// TIA Portal V17 program export: 0 tag tables, 0 data types, 22 data blocks, 121 code blocks (in call order from the OBs), 25 instance data blocks

DATA_BLOCK "Reminder"   // DB2
{ S7_Optimized_Access := 'TRUE' }
VERSION : 0.1
// stored: AutoNumber true, DBAccessibleFromOPCUA true, DBAccessibleFromWebserver true, IsOnlyStoredInLoadMemory false, IsRetainMemResEnabled false, IsWriteProtectedInAS false, MemoryReserve 100
   VAR
      x1 : Bool;
   END_VAR
BEGIN
END_DATA_BLOCK

DATA_BLOCK "HMI"   // DB110
{ S7_Optimized_Access := 'TRUE' }
VERSION : 0.1
// stored: AutoNumber false, DBAccessibleFromOPCUA true, DBAccessibleFromWebserver true, IsOnlyStoredInLoadMemory false, IsRetainMemResEnabled false, IsWriteProtectedInAS false, MemoryReserve 100
   VAR
      SS1 : Struct
         xLocalCmd : Bool;
         xEnbCmd : Bool := True;
         xLocalSt : Bool;
         rPacRef : Real;
         rQacRef : Real;
      END_STRUCT;
      SS2 : Struct
         xLocalCmd : Bool;
         xEnbCmd : Bool := True;
         xLocalSt : Bool;
         rPacRef : Real;
         rQacRef : Real;
      END_STRUCT;
      xLocalCmd : Bool;
      xStopCmd : Bool;
      xStandByCmd : Bool;
      xRunCmd : Bool;
      xTestCmd : Bool;
      xLocalSt : Bool;
      xStopSt : Bool;
      xStandBySt : Bool;
      xRunSt : Bool;
      rPacAutomRef : Real;
      PCS1 : Struct
         xEnbDCbus1 : Bool := True;
         xEnbDCbus2 : Bool := True;
      END_STRUCT;
      iNMaxRackFault : Int := 1;
      iNMinRackEnable : Int := 1;
      rSnPE : Real;
      xBB1BR1AlmDisable : Bool;
      xBB1BR2AlmDisable : Bool;
      xBB1BR3AlmDisable : Bool;
      xBB1BR4AlmDisable : Bool;
      xBB1BR5AlmDisable : Bool;
      xBB1BR6AlmDisable : Bool;
      xBB1BR7AlmDisable : Bool;
      xBB1BR8AlmDisable : Bool;
      xBB1BR9AlmDisable : Bool;
      xBB1BR10AlmDisable : Bool;
      xBB2BR1AlmDisable : Bool;
      xBB2BR2AlmDisable : Bool;
      xBB2BR3AlmDisable : Bool;
      xBB2BR4AlmDisable : Bool;
      xBB2BR5AlmDisable : Bool;
      xBB2BR6AlmDisable : Bool;
      xBB2BR7AlmDisable : Bool;
      xBB2BR8AlmDisable : Bool;
      xBB2BR9AlmDisable : Bool;
      xBB2BR10AlmDisable : Bool;
      xBB1AlmDisable : Bool;
      xBB2AlmDisable : Bool;
      xPEMSAlmDisable : Bool;
      xPCSAlmDisable : Bool;
      xMVSkidAlmDisable : Bool;
      xPIAlmDisable : Bool;
   END_VAR
BEGIN
END_DATA_BLOCK

DATA_BLOCK "SM_TEST"   // DB9
{ S7_Optimized_Access := 'TRUE' }
VERSION : 0.1
// stored: AutoNumber true, DBAccessibleFromOPCUA true, DBAccessibleFromWebserver true, IsOnlyStoredInLoadMemory false, IsRetainMemResEnabled false, IsWriteProtectedInAS false, MemoryReserve 100
   VAR
      xEnable_comm : Bool;
      xComm_enabled : Bool;
      xSS1_fault : Bool;
      xAutoCharge_command : Bool;
      xSM1_readyCondition : Bool;
      xSystem_ready : Bool;
      "xBattery_cl/op_command" : Bool;
      xBypass_Estop : Bool;
   END_VAR
BEGIN
END_DATA_BLOCK

DATA_BLOCK "clock"   // DB4
{ S7_Optimized_Access := 'TRUE' }
VERSION : 0.1
// stored: AutoNumber true, DBAccessibleFromOPCUA true, DBAccessibleFromWebserver true, IsOnlyStoredInLoadMemory false, IsRetainMemResEnabled false, IsWriteProtectedInAS false, MemoryReserve 100
   VAR
      xClock_5Hz : Bool;
      xClock_2_5Hz : Bool;
      xClock_2Hz : Bool;
      xClock_1_25Hz : Bool;
      xClock_1Hz : Bool;
      xClock_0_625Hz : Bool;
      xClock_0_5Hz : Bool;
      xClock_10Hz : Bool;
   END_VAR
BEGIN
END_DATA_BLOCK

DATA_BLOCK "BMS1"   // DB21
{ S7_Optimized_Access := 'TRUE' }
VERSION : 0.1
// stored: AutoNumber false, DBAccessibleFromOPCUA true, DBAccessibleFromWebserver true, IsOnlyStoredInLoadMemory false, IsRetainMemResEnabled false, IsWriteProtectedInAS false, MemoryReserve 100
   VAR RETAIN
      TCON { S7_SetPoint := 'True'} : TCON_IP_v4;
   END_VAR
   VAR
      arrData : Array[1..125] of Word;
      xREQ : Bool;
      iCountDone : Int := 1;
      iCountRead : Int := 1;
      MBmode : USInt;
      MBdataAddr : UDInt;
      MBdataLen : UInt;
   END_VAR
   VAR RETAIN
      TCON10 { S7_SetPoint := 'True'} : TCON_IP_v4;
   END_VAR
   VAR
      arrData10 : Array[1..125] of Word;
      xREQ10 : Bool;
      iCountDone10 : Int := 1;
      iCountRead10 : Int := 1;
      MBmode10 : USInt;
      MBdataAddr10 : UDInt;
      MBdataLen10 : UInt;
   END_VAR
   VAR RETAIN
      TCON11 { S7_SetPoint := 'True'} : TCON_IP_v4;
   END_VAR
   VAR
      arrData11 : Array[1..125] of Word;
      xREQ11 : Bool;
      iCountDone11 : Int := 1;
      iCountRead11 : Int := 1;
      MBmode11 : USInt;
      MBdataAddr11 : UDInt;
      MBdataLen11 : UInt;
      BB { S7_SetPoint := 'True'} : "BMS_BB";
      BR01 { S7_SetPoint := 'True'} : "BMS_BR";
      BR02 { S7_SetPoint := 'True'} : "BMS_BR";
      BR03 { S7_SetPoint := 'True'} : "BMS_BR";
      BR04 { S7_SetPoint := 'True'} : "BMS_BR";
      BR05 { S7_SetPoint := 'True'} : "BMS_BR";
      BR06 { S7_SetPoint := 'True'} : "BMS_BR";
      BR07 { S7_SetPoint := 'True'} : "BMS_BR";
      BR08 { S7_SetPoint := 'True'} : "BMS_BR";
      BR09 { S7_SetPoint := 'True'} : "BMS_BR";
      BR10 { S7_SetPoint := 'True'} : "BMS_BR";
      BR11 { S7_SetPoint := 'True'} : "BMS_BR";
      BR12 { S7_SetPoint := 'True'} : "BMS_BR";
      TMS01 { S7_SetPoint := 'True'} : "BMS_TMS";
      TMS02 { S7_SetPoint := 'True'} : "BMS_TMS";
      TMS03 { S7_SetPoint := 'True'} : "BMS_TMS";
      TMS04 { S7_SetPoint := 'True'} : "BMS_TMS";
      TMS05 { S7_SetPoint := 'True'} : "BMS_TMS";
      TMS06 { S7_SetPoint := 'True'} : "BMS_TMS";
      TMS07 { S7_SetPoint := 'True'} : "BMS_TMS";
      TMS08 { S7_SetPoint := 'True'} : "BMS_TMS";
      TMS09 { S7_SetPoint := 'True'} : "BMS_TMS";
      TMS10 { S7_SetPoint := 'True'} : "BMS_TMS";
      TMS11 { S7_SetPoint := 'True'} : "BMS_TMS";
      TMS12 { S7_SetPoint := 'True'} : "BMS_TMS";
      rNomEnergyBank { S7_SetPoint := 'True'} : Real;
      rPbank : Real;
      rCrate : Real;
      rSOCavlCha : Real;
      rSOCavlDsch : Real;
      rEnergyAvlCha : Real;
      rEnergyAvlDsch : Real;
      diTimeEndCha : DInt;
      diTimeEndDsch : DInt;
      rVcellMinSet : Real := 2.76;
      rVcellMinReset : Real := 3.05;
      rVcellMaxSet : Real := 3.68;
      rVcellMaxReset : Real := 3.3;
      rVcellAutoChaSet : Real := 2.7;
      rVcellAutoChaReset : Real := 3.1;
      rPchaLim : Real;
      rPdschLim : Real;
      wRackFlt : Word;
      wRackOn : Word;
      xBankAvl : Bool;
      xEnbCha : Bool;
      xEnbDsch : Bool;
      xAutoChaCmd : Bool;
      xSwitchGearSt : Bool;
      xPwrOffReadySt : Bool;
      xPwrOnReadySt : Bool;
      xPwrOnFltSt : Bool;
      xPwrOffFltSt : Bool;
      xInitSt : Bool;
      xNormOpSt : Bool;
      xFullChaSt : Bool;
      xFullDschSt : Bool;
      xWarnSt : Bool;
      xFltSt : Bool;
      xInitCmd : Bool;
      xStayCmd : Bool;
      xCloseCmd : Bool;
      xOpenCmd : Bool;
      xFltClearCmd : Bool;
      wCmd : Word;
      wFltClearCmd : Word;
      BBwAlm1 : Word;
      BBwWarn1 : Word;
      BBxCommFltSt : Bool;
      BBxFltSt : Bool;
      BBxAlmSt : Bool;
      BBxWarnSt : Bool;
      BR01wAlm1 : Word;
      BR01wAlm2 : Word;
      BR01wAlm3 : Word;
      BR01wWarn1 : Word;
      BR01xFltSt : Bool;
      BR01xAlmSt : Bool;
      BR01xWarnSt : Bool;
      BR02wAlm1 : Word;
      BR02wAlm2 : Word;
      BR02wAlm3 : Word;
      BR02wWarn1 : Word;
      BR02xFltSt : Bool;
      BR02xAlmSt : Bool;
      BR02xWarnSt : Bool;
      BR03wAlm1 : Word;
      BR03wAlm2 : Word;
      BR03wAlm3 : Word;
      BR03wWarn1 : Word;
      BR03xFltSt : Bool;
      BR03xAlmSt : Bool;
      BR03xWarnSt : Bool;
      BR04wAlm1 : Word;
      BR04wAlm2 : Word;
      BR04wAlm3 : Word;
      BR04wWarn1 : Word;
      BR04xFltSt : Bool;
      BR04xAlmSt : Bool;
      BR04xWarnSt : Bool;
      BR05wAlm1 : Word;
      BR05wAlm2 : Word;
      BR05wAlm3 : Word;
      BR05wWarn1 : Word;
      BR05xFltSt : Bool;
      BR05xAlmSt : Bool;
      BR05xWarnSt : Bool;
      BR06wAlm1 : Word;
      BR06wAlm2 : Word;
      BR06wAlm3 : Word;
      BR06wWarn1 : Word;
      BR06xFltSt : Bool;
      BR06xAlmSt : Bool;
      BR06xWarnSt : Bool;
      BR07wAlm1 : Word;
      BR07wAlm2 : Word;
      BR07wAlm3 : Word;
      BR07wWarn1 : Word;
      BR07xFltSt : Bool;
      BR07xAlmSt : Bool;
      BR07xWarnSt : Bool;
      BR08wAlm1 : Word;
      BR08wAlm2 : Word;
      BR08wAlm3 : Word;
      BR08wWarn1 : Word;
      BR08xFltSt : Bool;
      BR08xAlmSt : Bool;
      BR08xWarnSt : Bool;
      BR09wAlm1 : Word;
      BR09wAlm2 : Word;
      BR09wAlm3 : Word;
      BR09wWarn1 : Word;
      BR09xFltSt : Bool;
      BR09xAlmSt : Bool;
      BR09xWarnSt : Bool;
      BR10wAlm1 : Word;
      BR10wAlm2 : Word;
      BR10wAlm3 : Word;
      BR10wWarn1 : Word;
      BR10xFltSt : Bool;
      BR10xAlmSt : Bool;
      BR10xWarnSt : Bool;
      BR11wAlm1 : Word;
      BR11wAlm2 : Word;
      BR11wAlm3 : Word;
      BR11wWarn1 : Word;
      BR11xFltSt : Bool;
      BR11xAlmSt : Bool;
      BR11xWarnSt : Bool;
      BR12wAlm1 : Word;
      BR12wAlm2 : Word;
      BR12wAlm3 : Word;
      BR12wWarn1 : Word;
      BR12xFltSt : Bool;
      BR12xAlmSt : Bool;
      BR12xWarnSt : Bool;
      iNRackFault : Int;
      BR01xSSFltSt : Bool;
      BR02xSSFltSt : Bool;
      BR03xSSFltSt : Bool;
      BR04xSSFltSt : Bool;
      BR05xSSFltSt : Bool;
      BR06xSSFltSt : Bool;
      BR07xSSFltSt : Bool;
      BR08xSSFltSt : Bool;
      BR09xSSFltSt : Bool;
      BR10xSSFltSt : Bool;
      BR11xSSFltSt : Bool;
      BR12xSSFltSt : Bool;
   END_VAR
BEGIN
   TCON.RemoteAddress.ADDR[1] := 192;
   TCON.RemoteAddress.ADDR[2] := 168;
   TCON.RemoteAddress.ADDR[3] := 150;
   TCON.RemoteAddress.ADDR[4] := 44;
   TCON10.RemoteAddress.ADDR[1] := 192;
   TCON10.RemoteAddress.ADDR[2] := 168;
   TCON10.RemoteAddress.ADDR[3] := 150;
   TCON10.RemoteAddress.ADDR[4] := 44;
   TCON11.RemoteAddress.ADDR[1] := 192;
   TCON11.RemoteAddress.ADDR[2] := 168;
   TCON11.RemoteAddress.ADDR[3] := 150;
   TCON11.RemoteAddress.ADDR[4] := 44;
   BB.iNBRtotalCount := 10;
END_DATA_BLOCK

DATA_BLOCK "BMS2"   // DB22
{ S7_Optimized_Access := 'TRUE' }
VERSION : 0.1
// stored: AutoNumber false, DBAccessibleFromOPCUA true, DBAccessibleFromWebserver true, IsOnlyStoredInLoadMemory false, IsRetainMemResEnabled false, IsWriteProtectedInAS false, MemoryReserve 100
   VAR RETAIN
      TCON { S7_SetPoint := 'True'} : TCON_IP_v4;
   END_VAR
   VAR
      arrData : Array[1..125] of Word;
      xREQ : Bool;
      iCountDone : Int := 1;
      iCountRead : Int := 1;
      MBmode : USInt;
      MBdataAddr : UDInt;
      MBdataLen : UInt;
   END_VAR
   VAR RETAIN
      TCON10 { S7_SetPoint := 'True'} : TCON_IP_v4;
   END_VAR
   VAR
      arrData10 : Array[1..125] of Word;
      xREQ10 : Bool;
      iCountDone10 : Int := 1;
      iCountRead10 : Int := 1;
      MBmode10 : USInt;
      MBdataAddr10 : UDInt;
      MBdataLen10 : UInt;
   END_VAR
   VAR RETAIN
      TCON11 { S7_SetPoint := 'True'} : TCON_IP_v4;
   END_VAR
   VAR
      arrData11 : Array[1..125] of Word;
      xREQ11 : Bool;
      iCountDone11 : Int := 1;
      iCountRead11 : Int := 1;
      MBmode11 : USInt;
      MBdataAddr11 : UDInt;
      MBdataLen11 : UInt;
      BB { S7_SetPoint := 'True'} : "BMS_BB";
      BR01 { S7_SetPoint := 'True'} : "BMS_BR";
      BR02 { S7_SetPoint := 'True'} : "BMS_BR";
      BR03 { S7_SetPoint := 'True'} : "BMS_BR";
      BR04 { S7_SetPoint := 'True'} : "BMS_BR";
      BR05 { S7_SetPoint := 'True'} : "BMS_BR";
      BR06 { S7_SetPoint := 'True'} : "BMS_BR";
      BR07 { S7_SetPoint := 'True'} : "BMS_BR";
      BR08 { S7_SetPoint := 'True'} : "BMS_BR";
      BR09 { S7_SetPoint := 'True'} : "BMS_BR";
      BR10 { S7_SetPoint := 'True'} : "BMS_BR";
      TMS01 { S7_SetPoint := 'True'} : "BMS_TMS";
      TMS02 { S7_SetPoint := 'True'} : "BMS_TMS";
      TMS03 { S7_SetPoint := 'True'} : "BMS_TMS";
      TMS04 { S7_SetPoint := 'True'} : "BMS_TMS";
      TMS05 { S7_SetPoint := 'True'} : "BMS_TMS";
      TMS06 { S7_SetPoint := 'True'} : "BMS_TMS";
      TMS07 { S7_SetPoint := 'True'} : "BMS_TMS";
      TMS08 { S7_SetPoint := 'True'} : "BMS_TMS";
      TMS09 { S7_SetPoint := 'True'} : "BMS_TMS";
      TMS10 { S7_SetPoint := 'True'} : "BMS_TMS";
      rNomEnergyBank { S7_SetPoint := 'True'} : Real;
      rPbank : Real;
      rCrate : Real;
      rSOCavlCha : Real;
      rSOCavlDsch : Real;
      rEnergyAvlCha : Real;
      rEnergyAvlDsch : Real;
      diTimeEndCha : DInt;
      diTimeEndDsch : DInt;
      rVcellMinSet : Real := 2.76;
      rVcellMinReset : Real := 3.05;
      rVcellMaxSet : Real := 3.68;
      rVcellMaxReset : Real := 3.3;
      rVcellAutoChaSet : Real := 2.7;
      rVcellAutoChaReset : Real := 3.1;
      rPchaLim : Real;
      rPdschLim : Real;
      wRackFlt : Word;
      wRackOn : Word;
      xBankAvl : Bool;
      xEnbCha : Bool;
      xEnbDsch : Bool;
      xAutoChaCmd : Bool;
      xSwitchGearSt : Bool;
      xPwrOffReadySt : Bool;
      xPwrOnReadySt : Bool;
      xPwrOnFltSt : Bool;
      xPwrOffFltSt : Bool;
      xInitSt : Bool;
      xNormOpSt : Bool;
      xFullChaSt : Bool;
      xFullDschSt : Bool;
      xWarnSt : Bool;
      xFltSt : Bool;
      xInitCmd : Bool;
      xStayCmd : Bool;
      xCloseCmd : Bool;
      xOpenCmd : Bool;
      xFltClearCmd : Bool;
      wCmd : Word;
      wFltClearCmd : Word;
      BBwAlm1 : Word;
      BBwWarn1 : Word;
      BBxCommFltSt : Bool;
      BBxFltSt : Bool;
      BBxAlmSt : Bool;
      BBxWarnSt : Bool;
      BR01wAlm1 : Word;
      BR01wAlm2 : Word;
      BR01wAlm3 : Word;
      BR01wWarn1 : Word;
      BR01xFltSt : Bool;
      BR01xAlmSt : Bool;
      BR01xWarnSt : Bool;
      BR02wAlm1 : Word;
      BR02wAlm2 : Word;
      BR02wAlm3 : Word;
      BR02wWarn1 : Word;
      BR02xFltSt : Bool;
      BR02xAlmSt : Bool;
      BR02xWarnSt : Bool;
      BR03wAlm1 : Word;
      BR03wAlm2 : Word;
      BR03wAlm3 : Word;
      BR03wWarn1 : Word;
      BR03xFltSt : Bool;
      BR03xAlmSt : Bool;
      BR03xWarnSt : Bool;
      BR04wAlm1 : Word;
      BR04wAlm2 : Word;
      BR04wAlm3 : Word;
      BR04wWarn1 : Word;
      BR04xFltSt : Bool;
      BR04xAlmSt : Bool;
      BR04xWarnSt : Bool;
      BR05wAlm1 : Word;
      BR05wAlm2 : Word;
      BR05wAlm3 : Word;
      BR05wWarn1 : Word;
      BR05xFltSt : Bool;
      BR05xAlmSt : Bool;
      BR05xWarnSt : Bool;
      BR06wAlm1 : Word;
      BR06wAlm2 : Word;
      BR06wAlm3 : Word;
      BR06wWarn1 : Word;
      BR06xFltSt : Bool;
      BR06xAlmSt : Bool;
      BR06xWarnSt : Bool;
      BR07wAlm1 : Word;
      BR07wAlm2 : Word;
      BR07wAlm3 : Word;
      BR07wWarn1 : Word;
      BR07xFltSt : Bool;
      BR07xAlmSt : Bool;
      BR07xWarnSt : Bool;
      BR08wAlm1 : Word;
      BR08wAlm2 : Word;
      BR08wAlm3 : Word;
      BR08wWarn1 : Word;
      BR08xFltSt : Bool;
      BR08xAlmSt : Bool;
      BR08xWarnSt : Bool;
      BR09wAlm1 : Word;
      BR09wAlm2 : Word;
      BR09wAlm3 : Word;
      BR09wWarn1 : Word;
      BR09xFltSt : Bool;
      BR09xAlmSt : Bool;
      BR09xWarnSt : Bool;
      BR10wAlm1 : Word;
      BR10wAlm2 : Word;
      BR10wAlm3 : Word;
      BR10wWarn1 : Word;
      BR10xFltSt : Bool;
      BR10xAlmSt : Bool;
      BR10xWarnSt : Bool;
      iNRackFault : Int;
      BR01xSSFltSt : Bool;
      BR02xSSFltSt : Bool;
      BR03xSSFltSt : Bool;
      BR04xSSFltSt : Bool;
      BR05xSSFltSt : Bool;
      BR06xSSFltSt : Bool;
      BR07xSSFltSt : Bool;
      BR08xSSFltSt : Bool;
      BR09xSSFltSt : Bool;
      BR10xSSFltSt : Bool;
   END_VAR
BEGIN
   TCON.RemoteAddress.ADDR[1] := 192;
   TCON.RemoteAddress.ADDR[2] := 168;
   TCON.RemoteAddress.ADDR[3] := 150;
   TCON.RemoteAddress.ADDR[4] := 44;
   TCON10.RemoteAddress.ADDR[1] := 192;
   TCON10.RemoteAddress.ADDR[2] := 168;
   TCON10.RemoteAddress.ADDR[3] := 150;
   TCON10.RemoteAddress.ADDR[4] := 44;
   TCON11.RemoteAddress.ADDR[1] := 192;
   TCON11.RemoteAddress.ADDR[2] := 168;
   TCON11.RemoteAddress.ADDR[3] := 150;
   TCON11.RemoteAddress.ADDR[4] := 44;
   BB.iNBRtotalCount := 10;
END_DATA_BLOCK

DATA_BLOCK "EME"   // DB502, F_DB
{ S7_Optimized_Access := 'TRUE' }
VERSION : 0.1
// stored: AutoNumber false, DBAccessibleFromOPCUA true, DBAccessibleFromWebserver true
   VAR
      xAlwaysOff : Bool;
      xBattOpenCmd : Bool;
      xStopPCSCmd : Bool;
      xMVbrkOpenCmd : Bool;
      xMVtrafoSt : Bool;
      xAuxSkid : Bool;
      xAuxSkidDelay : Bool;
      xAuxSkidFireMan : Bool;
      xAuxSkidFireManDelay : Bool;
      xCore : Bool;
      xCoreDelay : Bool;
      xTwinPCS : Bool;
      xPCSCmd : Bool;
      xResetCmd : Bool;
      xByPass : Bool;
      xRcvError : Bool;
      xSendError : Bool;
      xAckReq : Bool;
      xByPassCore : Bool;
   END_VAR
BEGIN
END_DATA_BLOCK

DATA_BLOCK "Emergency_DB"   // DB502, F_DB
{ S7_Optimized_Access := 'TRUE' }
VERSION : 0.1
// stored: AutoNumber false, DBAccessibleFromOPCUA true, DBAccessibleFromWebserver true
   VAR
      xAlwaysOff : Bool;
      xBattOpenCmd : Bool;
      xStopPCSCmd : Bool;
      xMVbrkOpenCmd : Bool;
      xMVtrafoSt : Bool;
      xAuxSkid : Bool;
      xAuxSkidDelay : Bool;
      xAuxSkidFireMan : Bool;
      xAuxSkidFireManDelay : Bool;
      xCore : Bool;
      xCoreDelay : Bool;
      xTwinPCS : Bool;
      xPCSCmd : Bool;
      xResetCmd : Bool;
      xByPass : Bool;
      xRcvError : Bool;
      xSendError : Bool;
      xAckReq : Bool;
      xByPassCore : Bool;
      xTripPemsBattery : Bool;
   END_VAR
BEGIN
END_DATA_BLOCK

DATA_BLOCK "SM1"   // DB61
{ S7_Optimized_Access := 'TRUE' }
VERSION : 0.1
// stored: AutoNumber false, DBAccessibleFromOPCUA true, DBAccessibleFromWebserver true, IsOnlyStoredInLoadMemory false, IsRetainMemResEnabled false, IsWriteProtectedInAS false, MemoryReserve 100
   VAR
      xT11 : Bool;
      xT21 : Bool;
      xT22 : Bool;
      xT31 : Bool;
      xT32 : Bool;
      xT33 : Bool;
      xT34 : Bool;
      xT41 : Bool;
      xT42 : Bool;
      xT43 : Bool;
      xT44 : Bool;
      xT51 : Bool;
      xT52 : Bool;
      xT53 : Bool;
      xT61 : Bool;
      xT62 : Bool;
      xT71 : Bool;
      xT72 : Bool;
      xT73 : Bool;
      xT81 : Bool;
      xT91 : Bool;
      xSsBootSt : Bool;
      xSsWarmUpSt : Bool;
      xSsReadySt : Bool;
      xSsStandBySt : Bool;
      xSsRunSt : Bool;
      xSsTestSt : Bool;
      xSsAutoMaintSt : Bool;
      xSsStopSt : Bool;
      xSsFaultSt : Bool;
      iCountSS : Int;
      xBootSt : Bool;
      xRunPlcSt : Bool;
      xCommCmd : Bool;
      xAuxCmd : Bool;
      xCommSt : Bool;
      xAuxSt : Bool;
      xFltSt : Bool;
      xEnbSSysSt : Bool;
      xReadyCondSt : Bool;
      xTestCmd : Bool;
      xBattCloseCmd : Bool;
      xBattCloseSt : Bool;
      xBattOpenSt : Bool;
      xStopCmd : Bool;
      xStandByCmd : Bool;
      xAutomaintCmd : Bool;
      xStopAutomaintCmd : Bool;
      xAutomaintSt : Bool;
      xRunCmd : Bool;
      xPCSenbCmd : Bool;
      xPCSrunCmd : Bool;
      xMVbreakerCloseSt : Bool;
      xPCSrunSt : Bool;
      xPCSstopSt : Bool;
      xPCSreadySt : Bool;
      rPacAutomRef : Real;
      xVacPCS : Bool;
      xMVbreakerOpenCmd : Bool;
      xMVbreakerOpenSt : Bool;
   END_VAR
BEGIN
END_DATA_BLOCK

DATA_BLOCK "SM2"   // DB71
{ S7_Optimized_Access := 'TRUE' }
VERSION : 0.1
// stored: AutoNumber false, DBAccessibleFromOPCUA true, DBAccessibleFromWebserver true, IsOnlyStoredInLoadMemory false, IsRetainMemResEnabled false, IsWriteProtectedInAS false, MemoryReserve 100
   VAR
      xT11 : Bool;
      xT21 : Bool;
      xT22 : Bool;
      xT31 : Bool;
      xT32 : Bool;
      xT33 : Bool;
      xT34 : Bool;
      xT41 : Bool;
      xT42 : Bool;
      xT43 : Bool;
      xT44 : Bool;
      xT51 : Bool;
      xT52 : Bool;
      xT53 : Bool;
      xT61 : Bool;
      xT62 : Bool;
      xT71 : Bool;
      xT72 : Bool;
      xT73 : Bool;
      xT81 : Bool;
      xT91 : Bool;
      xSsBootSt : Bool;
      xSsWarmUpSt : Bool;
      xSsReadySt : Bool;
      xSsStandBySt : Bool;
      xSsRunSt : Bool;
      xSsTestSt : Bool;
      xSsAutoMaintSt : Bool;
      xSsStopSt : Bool;
      xSsFaultSt : Bool;
      iCountSS : Int;
      xBootSt : Bool;
      xRunPlcSt : Bool;
      xCommCmd : Bool;
      xAuxCmd : Bool;
      xCommSt : Bool;
      xAuxSt : Bool;
      xFltSt : Bool;
      xEnbSSysSt : Bool;
      xReadyCondSt : Bool;
      xTestCmd : Bool;
      xBattCloseCmd : Bool;
      xBattCloseSt : Bool;
      xBattOpenSt : Bool;
      xStopCmd : Bool;
      xStandByCmd : Bool;
      xAutomaintCmd : Bool;
      xStopAutomaintCmd : Bool;
      xAutomaintSt : Bool;
      xRunCmd : Bool;
      xPCSenbCmd : Bool;
      xPCSrunCmd : Bool;
      xMVbreakerCloseSt : Bool;
      xPCSrunSt : Bool;
      xPCSstopSt : Bool;
      xPCSreadySt : Bool;
      rPacAutomRef : Real;
      xVacPCS : Bool;
      xMVbreakerOpenCmd : Bool;
      xMVbreakerOpenSt : Bool;
   END_VAR
BEGIN
END_DATA_BLOCK

DATA_BLOCK "SS"   // DB101
{ S7_Optimized_Access := 'TRUE' }
VERSION : 0.1
// stored: AutoNumber false, DBAccessibleFromOPCUA true, DBAccessibleFromWebserver true, IsOnlyStoredInLoadMemory false, IsRetainMemResEnabled false, IsWriteProtectedInAS false, MemoryReserve 100
   VAR
      xFltSt : Bool;
      xSs1FltSt : Bool;
      xSs2FltSt : Bool;
      xAlmSt : Bool;
      XWarSt : Bool;   // Warning status
      wAlm1 : Word;
      wAlm2 : Word;
      wAlm3 : Word;
      wAlm4 : Word;
      wAlm5 : Word;
      wWarn1 : Word;
      wWarn2 : Word;
      wWarn3 : Word;
      wWarn4 : Word;
      wWarn5 : Word;
   END_VAR
BEGIN
END_DATA_BLOCK

DATA_BLOCK "DigitalOutput_DB"   // DB1
{ S7_Optimized_Access := 'TRUE' }
VERSION : 0.1
// stored: AutoNumber true, DBAccessibleFromOPCUA true, DBAccessibleFromWebserver true, IsOnlyStoredInLoadMemory false, IsRetainMemResEnabled false, IsWriteProtectedInAS false, MemoryReserve 100
   VAR
      xEnable : Bool;
   END_VAR
BEGIN
END_DATA_BLOCK

DATA_BLOCK "DashBoard"   // DB121
{ S7_Optimized_Access := 'FALSE' }
VERSION : 0.1
// stored: AutoNumber false, DBAccessibleFromOPCUA true, DBAccessibleFromWebserver true, IsOnlyStoredInLoadMemory false, IsWriteProtectedInAS false
   VAR
      BB1 { S7_SetPoint := 'True'} : "BB";
      BB2 { S7_SetPoint := 'True'} : "BB";
      BB1BR1 : "BR";
      BB1BR2 : "BR";
      BB1BR3 : "BR";
      BB1BR4 : "BR";
      BB1BR5 : "BR";
      BB1BR6 : "BR";
      BB1BR7 : "BR";
      BB1BR8 : "BR";
      BB1BR9 : "BR";
      BB1BR10 : "BR";
      BB1BR11 : "BR";
      BB1BR12 : "BR";
      BB2BR1 : "BR";
      BB2BR2 : "BR";
      BB2BR3 : "BR";
      BB2BR4 : "BR";
      BB2BR5 : "BR";
      BB2BR6 : "BR";
      BB2BR7 : "BR";
      BB2BR8 : "BR";
      BB2BR9 : "BR";
      BB2BR10 : "BR";
      BB2BR11 : "BR";
      BB2BR12 : "BR";
      PCS : "PCS";
      MVSKID { S7_SetPoint := 'True'} : "MVSKID";
      SM { S7_SetPoint := 'True'} : "SM";
   END_VAR
BEGIN
END_DATA_BLOCK

DATA_BLOCK "ED"   // DB400
{ S7_Optimized_Access := 'TRUE' }
VERSION : 0.1
// stored: AutoNumber false, DBAccessibleFromOPCUA true, DBAccessibleFromWebserver true, IsOnlyStoredInLoadMemory false, IsRetainMemResEnabled false, IsWriteProtectedInAS false, MemoryReserve 100
   VAR
      Pems : Struct
         LinkState : Array[1..52] of "LPNDR_typePortLinkState";
         X1 : Bool;
         X2 : Bool;
         X3 : Bool;
      END_STRUCT;
      ET200 : Struct
         LinkState : Array[1..52] of "LPNDR_typePortLinkState";
         X1 : Bool;
         X2 : Bool;
      END_STRUCT;
   END_VAR
BEGIN
END_DATA_BLOCK

DATA_BLOCK "NTPserver"   // DB122
{ S7_Optimized_Access := 'TRUE' }
VERSION : 0.1
// stored: AutoNumber false, DBAccessibleFromOPCUA true, DBAccessibleFromWebserver true, IsOnlyStoredInLoadMemory false, IsRetainMemResEnabled false, IsWriteProtectedInAS false, MemoryReserve 100
   VAR
      x_lEnable : Bool := true;
      i_Reference : USInt;
      dtl_Time : DTL;
      i_auxRetVal : Int;
   END_VAR
BEGIN
END_DATA_BLOCK

DATA_BLOCK "MV SKID"   // DB42
{ S7_Optimized_Access := 'TRUE' }
VERSION : 0.1
// stored: AutoNumber false, DBAccessibleFromOPCUA true, DBAccessibleFromWebserver true, IsOnlyStoredInLoadMemory false, IsRetainMemResEnabled false, IsWriteProtectedInAS false, MemoryReserve 100
   VAR RETAIN
      TCON { S7_SetPoint := 'True'} : TCON_IP_v4;
   END_VAR
   VAR
      arrData : Array[1..125] of Word;
      xREQ : Bool;
      iCountDone : Int := 1;
      iCountRead : Int := 1;
      MBmode : USInt;
      MBdataAddr : UDInt;
      MBdataLen : UInt;
      R : "R_MV";
      W { S7_SetPoint := 'True'} : "W_MV";
      xFltSt { S7_SetPoint := 'True'} : Bool;
      xAlmSt : Bool;
      xWarnSt : Bool;
      wLine1DiscSt : Word;
      wLine2DiscSt : Word;
      wProt1DiscSt : Word;
      wProt1CircBrkSt : Word;
   END_VAR
BEGIN
   TCON.RemoteAddress.ADDR[1] := 192;
   TCON.RemoteAddress.ADDR[2] := 168;
   TCON.RemoteAddress.ADDR[3] := 150;
   TCON.RemoteAddress.ADDR[4] := 44;
END_DATA_BLOCK

DATA_BLOCK "MvSkid_1"   // DB42
{ S7_Optimized_Access := 'TRUE' }
VERSION : 0.1
// stored: AutoNumber false, DBAccessibleFromOPCUA true, DBAccessibleFromWebserver true, IsOnlyStoredInLoadMemory false, IsRetainMemResEnabled false, IsWriteProtectedInAS false, MemoryReserve 100
   VAR RETAIN
      TCON { S7_SetPoint := 'True'} : TCON_IP_v4;
   END_VAR
   VAR
      arrData : Array[1..125] of Word;
      xREQ : Bool;
      iCountRead : Int := 1;
      MBmode : USInt;
      MBdataAddr : UDInt;
      MBdataLen : UInt;
      R : "R_MV";
      iCountDone : Int := 1;
      W { S7_SetPoint := 'True'} : "W_MV";
      xFltSt { S7_SetPoint := 'True'} : Bool;
      xAlmSt : Bool;
      xWarnSt : Bool;
      wLine1DiscSt : Word;
      wLine2DiscSt : Word;
      wProt1DiscSt : Word;
      wProt1CircBrkSt : Word;
   END_VAR
BEGIN
   TCON.RemoteAddress.ADDR[1] := 192;
   TCON.RemoteAddress.ADDR[2] := 168;
   TCON.RemoteAddress.ADDR[3] := 150;
   TCON.RemoteAddress.ADDR[4] := 44;
END_DATA_BLOCK

DATA_BLOCK "MvSkid_2"   // DB46
{ S7_Optimized_Access := 'TRUE' }
VERSION : 0.1
// stored: AutoNumber true, DBAccessibleFromOPCUA true, DBAccessibleFromWebserver true, IsOnlyStoredInLoadMemory false, IsRetainMemResEnabled false, IsWriteProtectedInAS false, MemoryReserve 100
   VAR RETAIN
      TCON { S7_SetPoint := 'True'} : TCON_IP_v4;
   END_VAR
   VAR
      arrData : Array[1..125] of Word;
      xREQ : Bool;
      iCountDone : Int := 1;
      iCountRead : Int := 1;
      MBmode : USInt;
      MBdataAddr : UDInt;
      MBdataLen : UInt;
      R : "R_MV";
      W { S7_SetPoint := 'True'} : "W_MV";
      xFltSt { S7_SetPoint := 'True'} : Bool;
      xAlmSt : Bool;
      xWarnSt : Bool;
      wLine1DiscSt : Word;
      wLine2DiscSt : Word;
      wProt1DiscSt : Word;
      wProt1CircBrkSt : Word;
   END_VAR
BEGIN
   TCON.RemoteAddress.ADDR[1] := 192;
   TCON.RemoteAddress.ADDR[2] := 168;
   TCON.RemoteAddress.ADDR[3] := 150;
   TCON.RemoteAddress.ADDR[4] := 44;
END_DATA_BLOCK

DATA_BLOCK "PCS1"   // DB41
{ S7_Optimized_Access := 'TRUE' }
VERSION : 0.1
// stored: AutoNumber false, DBAccessibleFromOPCUA true, DBAccessibleFromWebserver true, IsOnlyStoredInLoadMemory false, IsRetainMemResEnabled false, IsWriteProtectedInAS false, MemoryReserve 100
   VAR RETAIN
      TCON { S7_SetPoint := 'True'} : TCON_IP_v4;
   END_VAR
   VAR
      arrData : Array[1..125] of Word;
      xREQ : Bool;
      iCountDone : Int := 1;
      iCountRead : Int := 1;
      MBmode : USInt;
      MBdataAddr : UDInt;
      MBdataLen : UInt;
   END_VAR
   VAR RETAIN
      TCON10 { S7_SetPoint := 'True'} : TCON_IP_v4;
   END_VAR
   VAR
      arrData10 : Array[1..125] of Word;
      xREQ10 : Bool;
      iCountDone10 : Int := 1;
      iCountRead10 : Int := 1;
      MBmode10 : USInt;
      MBdataAddr10 : UDInt;
      MBdataLen10 : UInt;
      R { S7_SetPoint := 'True'} : "R_PE";
      RW { S7_SetPoint := 'True'} : "RW_PE";
      W { S7_SetPoint := 'True'} : "W_PE";
   END_VAR
   VAR RETAIN
      TCONW { S7_SetPoint := 'True'} : TCON_IP_v4;
   END_VAR
   VAR
      arrDataW : Array[1..125] of Word;
      xREQW : Bool;
      iCountDoneW : Int := 1;
      iCountReadW : Int := 1;
      MBmodeW : USInt;
      MBdataAddrW : UDInt;
      MBdataLenW : UInt;
      xDCbus1Avl : Bool;
      xDCbus2Avl : Bool;
      xLVRT : Bool;
      xOVRT : Bool;
      xCommFltSt : Bool;
      xFltSt : Bool;
      xWarnSt : Bool;
      xModFltBus1St : Bool;
      xModFltBus2St : Bool;
      xMod1FltSt : Bool;
      xMod2FltSt : Bool;
      xMod3FltSt : Bool;
      xMod4FltSt : Bool;
      xMod5FltSt : Bool;
      xMod6FltSt : Bool;
      xMod1WarnSt : Bool;
      xMod2WarnSt : Bool;
      xMod3WarnSt : Bool;
      xMod4WarnSt : Bool;
      xMod5WarnSt : Bool;
      xMod6WarnSt : Bool;
      rMod1MaxTemp : Real;
      rMod2MaxTemp : Real;
      rMod3MaxTemp : Real;
      rMod4MaxTemp : Real;
      rMod5MaxTemp : Real;
      rMod6MaxTemp : Real;
      rPacBus1Meas : Real;
      rPacBus2Meas : Real;
      rQacBus1Meas : Real;
      rQacBus2Meas : Real;
      rVacMeas : Real;
      rIacTotMeas : Real;
      iCodeFlt : Int;
      iCodeWarn : Int;
      iModFlt : Int;
      iModWarn : Int;
      wInvFlt1 : Word;
      wInvFlt2 : Word;
      wInvFlt3 : Word;
      wInvFlt4 : Word;
      wInvFlt5 : Word;
      wInvFlt6 : Word;
      wInvFlt7 : Word;
      wInvWarn1 : Word;
      wInvWarn2 : Word;
      wInvWarn3 : Word;
      wInvWarn4 : Word;
      wInvWarn5 : Word;
      wInvWarn6 : Word;
      wMod1Flt1 : Word;
      wMod1Flt2 : Word;
      wMod1Flt3 : Word;
      wMod1Flt4 : Word;
      wMod2Flt1 : Word;
      wMod2Flt2 : Word;
      wMod2Flt3 : Word;
      wMod2Flt4 : Word;
      wMod3Flt1 : Word;
      wMod3Flt2 : Word;
      wMod3Flt3 : Word;
      wMod3Flt4 : Word;
      wMod4Flt1 : Word;
      wMod4Flt2 : Word;
      wMod4Flt3 : Word;
      wMod4Flt4 : Word;
      wMod5Flt1 : Word;
      wMod5Flt2 : Word;
      wMod5Flt3 : Word;
      wMod5Flt4 : Word;
      wMod6Flt1 : Word;
      wMod6Flt2 : Word;
      wMod6Flt3 : Word;
      wMod6Flt4 : Word;
      wMod1Warn1 : Word;
      wMod1Warn2 : Word;
      wMod1Warn3 : Word;
      wMod1Warn4 : Word;
      wMod2Warn1 : Word;
      wMod2Warn2 : Word;
      wMod2Warn3 : Word;
      wMod2Warn4 : Word;
      wMod3Warn1 : Word;
      wMod3Warn2 : Word;
      wMod3Warn3 : Word;
      wMod3Warn4 : Word;
      wMod4Warn1 : Word;
      wMod4Warn2 : Word;
      wMod4Warn3 : Word;
      wMod4Warn4 : Word;
      wMod5Warn1 : Word;
      wMod5Warn2 : Word;
      wMod5Warn3 : Word;
      wMod5Warn4 : Word;
      wMod6Warn1 : Word;
      wMod6Warn2 : Word;
      wMod6Warn3 : Word;
      wMod6Warn4 : Word;
      aWbit : Struct
         xStart : Word;
         xStopW : Word;
         xResetW : Word;
         xEnableW : Word;
         xEmergency : Word;
      END_STRUCT;
   END_VAR
BEGIN
   TCON.RemoteAddress.ADDR[1] := 192;
   TCON.RemoteAddress.ADDR[2] := 168;
   TCON.RemoteAddress.ADDR[3] := 150;
   TCON.RemoteAddress.ADDR[4] := 44;
   TCON10.RemoteAddress.ADDR[1] := 192;
   TCON10.RemoteAddress.ADDR[2] := 168;
   TCON10.RemoteAddress.ADDR[3] := 150;
   TCON10.RemoteAddress.ADDR[4] := 44;
   TCONW.RemoteAddress.ADDR[1] := 192;
   TCONW.RemoteAddress.ADDR[2] := 168;
   TCONW.RemoteAddress.ADDR[3] := 150;
   TCONW.RemoteAddress.ADDR[4] := 44;
END_DATA_BLOCK

DATA_BLOCK "PCS_1"   // DB41
{ S7_Optimized_Access := 'TRUE' }
VERSION : 0.1
// stored: AutoNumber false, DBAccessibleFromOPCUA true, DBAccessibleFromWebserver true, IsOnlyStoredInLoadMemory false, IsRetainMemResEnabled false, IsWriteProtectedInAS false, MemoryReserve 100
   VAR RETAIN
      TCONR_slow { S7_SetPoint := 'True'} : TCON_IP_v4;
   END_VAR
   VAR
      arrDataR_slow : Array[1..125] of Word;
      xREQR_slow : Bool;
      iCountDoneR_slow : Int := 1;
      iCountReadR_slow : Int := 1;
      MBmodeR_slow : USInt;
      MBdataAddrR_slow : UDInt;
      MBdataLenR_slow : UInt;
   END_VAR
   VAR RETAIN
      TCONR_fast { S7_SetPoint := 'True'} : TCON_IP_v4;
   END_VAR
   VAR
      arrDataR_fast : Array[1..125] of Word;
      xREQR_fast : Bool;
      iCountDoneR_fast : Int := 1;
      iCountReadR_fast : Int := 1;
      MBmodeR_fast : USInt;
      MBdataAddrR_fast : UDInt;
      MBdataLenR_fast : UInt;
   END_VAR
   VAR RETAIN
      TCONW_slow { S7_SetPoint := 'True'} : TCON_IP_v4;
   END_VAR
   VAR
      arrDataW_slow : Array[1..125] of Word;
      xREQW_slow : Bool;
      iCountDoneW_slow : Int := 1;
      iCountReadW_slow : Int := 1;
      MBmodeW_slow : USInt;
      MBdataAddrW_slow : UDInt;
      MBdataLenW_slow : UInt;
   END_VAR
   VAR RETAIN
      TCONW_fast { S7_SetPoint := 'True'} : TCON_IP_v4;
   END_VAR
   VAR
      arrDataW_fast : Array[1..125] of Word;
      xREQW_fast : Bool;
      iCountDoneW_fast : Int := 1;
      iCountReadW_fast : Int := 1;
      MBmodeW_fast : USInt;
      MBdataAddrW_fast : UDInt;
      MBdataLenW_fast : UInt;
      "____FINE SEGNALI CLIENT_____" : UInt;
      R { S7_SetPoint := 'True'} : "R_PE";
      RW { S7_SetPoint := 'True'} : "RW_PE";
      W { S7_SetPoint := 'True'} : "W_PE";
      arrStatus { S7_SetPoint := 'True'} : Array[0..17] of Bool;
      xDCbusAvl : Bool;
      xLVRT : Bool;
      xOVRT : Bool;
      xCommFltSt : Bool;
      xFltSt : Bool;
      xWarnSt : Bool;
      xModFltBus1St : Bool;
      xModFltBus2St : Bool;
      xMod1FltSt : Bool;
      xMod2FltSt : Bool;
      xMod3FltSt : Bool;
      xMod4FltSt : Bool;
      xMod5FltSt : Bool;
      xMod6FltSt : Bool;
      xMod1WarnSt : Bool;
      xMod2WarnSt : Bool;
      xMod3WarnSt : Bool;
      xMod4WarnSt : Bool;
      xMod5WarnSt : Bool;
      xMod6WarnSt : Bool;
      rMod1MaxTemp : Real;
      rMod2MaxTemp : Real;
      rMod3MaxTemp : Real;
      rMod4MaxTemp : Real;
      rMod5MaxTemp : Real;
      rMod6MaxTemp : Real;
      rPacBus1Meas : Real;
      rPacBus2Meas : Real;
      rQacBus1Meas : Real;
      rQacBus2Meas : Real;
      rLVacMeas : Real;
      rMVacMeas : Real;
      rIacTotMeas : Real;
      iCodeFlt : Int;
      iCodeWarn : Int;
      iModFlt : Int;
      iModWarn : Int;
      iLVac_Treshold : Int := 600;
      "____INVERTER FAULTS____" : Int;
      wInvFlt1 : Word;
      wInvFlt2 : Word;
      wInvFlt3 : Word;
      wInvFlt4 : Word;
      wInvFlt5 : Word;
      wInvFlt6 : Word;
      wInvFlt7 : Word;
      wInvWarn1 : Word;
      wInvWarn2 : Word;
      wInvWarn3 : Word;
      wInvWarn4 : Word;
      wInvWarn5 : Word;
      wInvWarn6 : Word;
      wMod1Flt1 : Word;
      wMod1Flt2 : Word;
      wMod1Flt3 : Word;
      wMod1Flt4 : Word;
      wMod2Flt1 : Word;
      wMod2Flt2 : Word;
      wMod2Flt3 : Word;
      wMod2Flt4 : Word;
      wMod3Flt1 : Word;
      wMod3Flt2 : Word;
      wMod3Flt3 : Word;
      wMod3Flt4 : Word;
      wMod4Flt1 : Word;
      wMod4Flt2 : Word;
      wMod4Flt3 : Word;
      wMod4Flt4 : Word;
      wMod5Flt1 : Word;
      wMod5Flt2 : Word;
      wMod5Flt3 : Word;
      wMod5Flt4 : Word;
      wMod6Flt1 : Word;
      wMod6Flt2 : Word;
      wMod6Flt3 : Word;
      wMod6Flt4 : Word;
      wMod1Warn1 : Word;
      wMod1Warn2 : Word;
      wMod1Warn3 : Word;
      wMod1Warn4 : Word;
      wMod2Warn1 : Word;
      wMod2Warn2 : Word;
      wMod2Warn3 : Word;
      wMod2Warn4 : Word;
      wMod3Warn1 : Word;
      wMod3Warn2 : Word;
      wMod3Warn3 : Word;
      wMod3Warn4 : Word;
      wMod4Warn1 : Word;
      wMod4Warn2 : Word;
      wMod4Warn3 : Word;
      wMod4Warn4 : Word;
      wMod5Warn1 : Word;
      wMod5Warn2 : Word;
      wMod5Warn3 : Word;
      wMod5Warn4 : Word;
      wMod6Warn1 : Word;
      wMod6Warn2 : Word;
      wMod6Warn3 : Word;
      wMod6Warn4 : Word;
      "_____TEST SIGNALS______" : Bool;
      xTestCmd : Bool;
      xTestRunCmd : Bool;
      xTestStopCmd : Bool;
      xTestResetCmd : Bool;
      xTestEnableCmd : Bool;
      xTestEmeCmd : Bool;
      "____SIGNAL EDGE______" : Bool;
      PSE : Struct
         x1 : Bool;
         x2 : Bool;
         x3 : Bool;
         x4 : Bool;
         x5 : Bool;
         x6 : Bool;
         x7 : Bool;
         x8 : Bool;
         x9 : Bool;
         x10 : Bool;
      END_STRUCT;
      NSE : Struct
         x1 : Bool;
         x2 : Bool;
         x3 : Bool;
         x4 : Bool;
         x5 : Bool;
         x6 : Bool;
         x7 : Bool;
         x8 : Bool;
         x9 : Bool;
         x10 : Bool;
      END_STRUCT;
   END_VAR
BEGIN
   TCONR_slow.RemoteAddress.ADDR[1] := 192;
   TCONR_slow.RemoteAddress.ADDR[2] := 168;
   TCONR_slow.RemoteAddress.ADDR[3] := 150;
   TCONR_slow.RemoteAddress.ADDR[4] := 44;
   TCONR_fast.RemoteAddress.ADDR[1] := 192;
   TCONR_fast.RemoteAddress.ADDR[2] := 168;
   TCONR_fast.RemoteAddress.ADDR[3] := 150;
   TCONR_fast.RemoteAddress.ADDR[4] := 44;
   // TCONW_slow.InterfaceId : HW_slow-identifier of IE-interface submodule
   TCONW_slow.RemoteAddress.ADDR[1] := 192;
   TCONW_slow.RemoteAddress.ADDR[2] := 168;
   TCONW_slow.RemoteAddress.ADDR[3] := 150;
   TCONW_slow.RemoteAddress.ADDR[4] := 44;
   TCONW_fast.RemoteAddress.ADDR[1] := 192;
   TCONW_fast.RemoteAddress.ADDR[2] := 168;
   TCONW_fast.RemoteAddress.ADDR[3] := 150;
   TCONW_fast.RemoteAddress.ADDR[4] := 44;
   // R.iCurrentStatus : Register 41004| 0:power up; 1:init; 2:off; 3:stanby DC; 4:precharge DC; 5:softcharge DC; 6:ready DC; 7:standby DC; 8:blackstart; 9:ready; 10:wait; 11:pre on; 12:on; 13:stop; 14:ready AC; 15:diagnostic AC; 16:discharge; 17:fault;
   // arrStatus[0] : power up
   // arrStatus[1] : init
   // arrStatus[2] : off
   // arrStatus[3] : standby DC
   // arrStatus[4] : precharge DC
   // arrStatus[5] : softcharge DC
   // arrStatus[6] : ready DC
   // arrStatus[7] : standby AC
   // arrStatus[8] : blackstart
   // arrStatus[9] : ready
   // arrStatus[10] : wait
   // arrStatus[11] : pre on
   // arrStatus[12] : on
   // arrStatus[13] : stop
   // arrStatus[14] : ready AC
   // arrStatus[15] : diagnostic AC
   // arrStatus[16] : discharge
   // arrStatus[17] : fault
END_DATA_BLOCK

DATA_BLOCK "PCS_2"   // DB43
{ S7_Optimized_Access := 'TRUE' }
VERSION : 0.1
// stored: AutoNumber true, DBAccessibleFromOPCUA true, DBAccessibleFromWebserver true, IsOnlyStoredInLoadMemory false, IsRetainMemResEnabled false, IsWriteProtectedInAS false, MemoryReserve 100
   VAR RETAIN
      TCONR_slow { S7_SetPoint := 'True'} : TCON_IP_v4;
   END_VAR
   VAR
      arrDataR_slow : Array[1..125] of Word;
      xREQR_slow : Bool;
      iCountDoneR_slow : Int := 1;
      iCountReadR_slow : Int := 1;
      MBmodeR_slow : USInt;
      MBdataAddrR_slow : UDInt;
      MBdataLenR_slow : UInt;
   END_VAR
   VAR RETAIN
      TCONR_fast { S7_SetPoint := 'True'} : TCON_IP_v4;
   END_VAR
   VAR
      arrDataR_fast : Array[1..125] of Word;
      xREQR_fast : Bool;
      iCountDoneR_fast : Int := 1;
      iCountReadR_fast : Int := 1;
      MBmodeR_fast : USInt;
      MBdataAddrR_fast : UDInt;
      MBdataLenR_fast : UInt;
   END_VAR
   VAR RETAIN
      TCONW_slow { S7_SetPoint := 'True'} : TCON_IP_v4;
   END_VAR
   VAR
      arrDataW_slow : Array[1..125] of Word;
      xREQW_slow : Bool;
      iCountDoneW_slow : Int := 1;
      iCountReadW_slow : Int := 1;
      MBmodeW_slow : USInt;
      MBdataAddrW_slow : UDInt;
      MBdataLenW_slow : UInt;
   END_VAR
   VAR RETAIN
      TCONW_fast { S7_SetPoint := 'True'} : TCON_IP_v4;
   END_VAR
   VAR
      arrDataW_fast : Array[1..125] of Word;
      xREQW_fast : Bool;
      iCountDoneW_fast : Int := 1;
      iCountReadW_fast : Int := 1;
      MBmodeW_fast : USInt;
      MBdataAddrW_fast : UDInt;
      MBdataLenW_fast : UInt;
      "____FINE SEGNALI CLIENT_____" : UInt;
      R { S7_SetPoint := 'True'} : "R_PE";
      RW { S7_SetPoint := 'True'} : "RW_PE";
      W { S7_SetPoint := 'True'} : "W_PE";
      arrStatus { S7_SetPoint := 'True'} : Array[0..17] of Bool;
      xDCbusAvl : Bool;
      xLVRT : Bool;
      xOVRT : Bool;
      xCommFltSt : Bool;
      xFltSt : Bool;
      xWarnSt : Bool;
      xModFltBus1St : Bool;
      xModFltBus2St : Bool;
      xMod1FltSt : Bool;
      xMod2FltSt : Bool;
      xMod3FltSt : Bool;
      xMod4FltSt : Bool;
      xMod5FltSt : Bool;
      xMod6FltSt : Bool;
      xMod1WarnSt : Bool;
      xMod2WarnSt : Bool;
      xMod3WarnSt : Bool;
      xMod4WarnSt : Bool;
      xMod5WarnSt : Bool;
      xMod6WarnSt : Bool;
      rMod1MaxTemp : Real;
      rMod2MaxTemp : Real;
      rMod3MaxTemp : Real;
      rMod4MaxTemp : Real;
      rMod5MaxTemp : Real;
      rMod6MaxTemp : Real;
      rPacBus1Meas : Real;
      rPacBus2Meas : Real;
      rQacBus1Meas : Real;
      rQacBus2Meas : Real;
      rLVacMeas : Real;
      rMVacMeas : Real;
      rIacTotMeas : Real;
      iCodeFlt : Int;
      iCodeWarn : Int;
      iModFlt : Int;
      iModWarn : Int;
      iLVac_Treshold : Int := 600;
      "____INVERTER FAULTS____" : Int;
      wInvFlt1 : Word;
      wInvFlt2 : Word;
      wInvFlt3 : Word;
      wInvFlt4 : Word;
      wInvFlt5 : Word;
      wInvFlt6 : Word;
      wInvFlt7 : Word;
      wInvWarn1 : Word;
      wInvWarn2 : Word;
      wInvWarn3 : Word;
      wInvWarn4 : Word;
      wInvWarn5 : Word;
      wInvWarn6 : Word;
      wMod1Flt1 : Word;
      wMod1Flt2 : Word;
      wMod1Flt3 : Word;
      wMod1Flt4 : Word;
      wMod2Flt1 : Word;
      wMod2Flt2 : Word;
      wMod2Flt3 : Word;
      wMod2Flt4 : Word;
      wMod3Flt1 : Word;
      wMod3Flt2 : Word;
      wMod3Flt3 : Word;
      wMod3Flt4 : Word;
      wMod4Flt1 : Word;
      wMod4Flt2 : Word;
      wMod4Flt3 : Word;
      wMod4Flt4 : Word;
      wMod5Flt1 : Word;
      wMod5Flt2 : Word;
      wMod5Flt3 : Word;
      wMod5Flt4 : Word;
      wMod6Flt1 : Word;
      wMod6Flt2 : Word;
      wMod6Flt3 : Word;
      wMod6Flt4 : Word;
      wMod1Warn1 : Word;
      wMod1Warn2 : Word;
      wMod1Warn3 : Word;
      wMod1Warn4 : Word;
      wMod2Warn1 : Word;
      wMod2Warn2 : Word;
      wMod2Warn3 : Word;
      wMod2Warn4 : Word;
      wMod3Warn1 : Word;
      wMod3Warn2 : Word;
      wMod3Warn3 : Word;
      wMod3Warn4 : Word;
      wMod4Warn1 : Word;
      wMod4Warn2 : Word;
      wMod4Warn3 : Word;
      wMod4Warn4 : Word;
      wMod5Warn1 : Word;
      wMod5Warn2 : Word;
      wMod5Warn3 : Word;
      wMod5Warn4 : Word;
      wMod6Warn1 : Word;
      wMod6Warn2 : Word;
      wMod6Warn3 : Word;
      wMod6Warn4 : Word;
      "_____TEST SIGNALS______" : Bool;
      xTestCmd : Bool;
      xTestRunCmd : Bool;
      xTestStopCmd : Bool;
      xTestResetCmd : Bool;
      xTestEnableCmd : Bool;
      xTestEmeCmd : Bool;
      "____SIGNAL EDGE______" : Bool;
      PSE : Struct
         x1 : Bool;
         x2 : Bool;
         x3 : Bool;
         x4 : Bool;
         x5 : Bool;
         x6 : Bool;
         x7 : Bool;
         x8 : Bool;
         x9 : Bool;
         x10 : Bool;
      END_STRUCT;
      NSE : Struct
         x1 : Bool;
         x2 : Bool;
         x3 : Bool;
         x4 : Bool;
         x5 : Bool;
         x6 : Bool;
         x7 : Bool;
         x8 : Bool;
         x9 : Bool;
         x10 : Bool;
      END_STRUCT;
   END_VAR
BEGIN
   TCONR_slow.RemoteAddress.ADDR[1] := 192;
   TCONR_slow.RemoteAddress.ADDR[2] := 168;
   TCONR_slow.RemoteAddress.ADDR[3] := 150;
   TCONR_slow.RemoteAddress.ADDR[4] := 44;
   TCONR_fast.RemoteAddress.ADDR[1] := 192;
   TCONR_fast.RemoteAddress.ADDR[2] := 168;
   TCONR_fast.RemoteAddress.ADDR[3] := 150;
   TCONR_fast.RemoteAddress.ADDR[4] := 44;
   // TCONW_slow.InterfaceId : HW_slow-identifier of IE-interface submodule
   TCONW_slow.RemoteAddress.ADDR[1] := 192;
   TCONW_slow.RemoteAddress.ADDR[2] := 168;
   TCONW_slow.RemoteAddress.ADDR[3] := 150;
   TCONW_slow.RemoteAddress.ADDR[4] := 44;
   TCONW_fast.RemoteAddress.ADDR[1] := 192;
   TCONW_fast.RemoteAddress.ADDR[2] := 168;
   TCONW_fast.RemoteAddress.ADDR[3] := 150;
   TCONW_fast.RemoteAddress.ADDR[4] := 44;
   // R.iCurrentStatus : Register 41004| 0:power up; 1:init; 2:off; 3:stanby DC; 4:precharge DC; 5:softcharge DC; 6:ready DC; 7:standby DC; 8:blackstart; 9:ready; 10:wait; 11:pre on; 12:on; 13:stop; 14:ready AC; 15:diagnostic AC; 16:discharge; 17:fault;
   // arrStatus[0] : power up
   // arrStatus[1] : init
   // arrStatus[2] : off
   // arrStatus[3] : standby DC
   // arrStatus[4] : precharge DC
   // arrStatus[5] : softcharge DC
   // arrStatus[6] : ready DC
   // arrStatus[7] : standby AC
   // arrStatus[8] : blackstart
   // arrStatus[9] : ready
   // arrStatus[10] : wait
   // arrStatus[11] : pre on
   // arrStatus[12] : on
   // arrStatus[13] : stop
   // arrStatus[14] : ready AC
   // arrStatus[15] : diagnostic AC
   // arrStatus[16] : discharge
   // arrStatus[17] : fault
END_DATA_BLOCK

DATA_BLOCK "PN"   // DB11
{ S7_Optimized_Access := 'TRUE' }
VERSION : 0.1
// stored: AutoNumber false, DBAccessibleFromOPCUA true, DBAccessibleFromWebserver true, IsOnlyStoredInLoadMemory false, IsRetainMemResEnabled false, IsWriteProtectedInAS false, MemoryReserve 100
   VAR
      DevOk : Array[0..1023] of Bool;
      FltDev : Array[0..1023] of Bool;
      R : "PN Read";
      W { S7_SetPoint := 'True'} : "PN Write";
      RV_R { S7_SetPoint := 'True'} : Int;
      RV_W { S7_SetPoint := 'True'} : Int;
      xStopCmd : Bool;
      xStandByCmd : Bool;
      xRunCmd : Bool;
      xFltCmd : Bool;
      xFltClearCmd : Bool;
      iKeepAlive : Int;
      SS1 : Struct
         rPacRef : Real;
         rQacRef : Real;
      END_STRUCT;
      SS2 : Struct
         rPacRef : Real;
         rQacRef : Real;
      END_STRUCT;
      MVSKID : Struct
         xCircBrkCloseCmd : Bool;
         xCircBrkOpenCmd : Bool;
      END_STRUCT;
   END_VAR
BEGIN
END_DATA_BLOCK

ORGANIZATION_BLOCK "Main"   // OB1, LAD, ProgramCycle
TITLE = "Main Program Sweep (Cycle)"
{ S7_Optimized_Access := 'TRUE' }
VERSION : 0.1
// stored: AutoNumber true, IsIECCheckEnabled false, SetENOAutomatically false
   VAR_INPUT
      Initial_Call : Bool;   // Initial call of this OB
      Remanence : Bool;   // =True, if remanent data are available
   END_VAR
BEGIN

REGION Network 1: Acknowledgement ProfiSafe
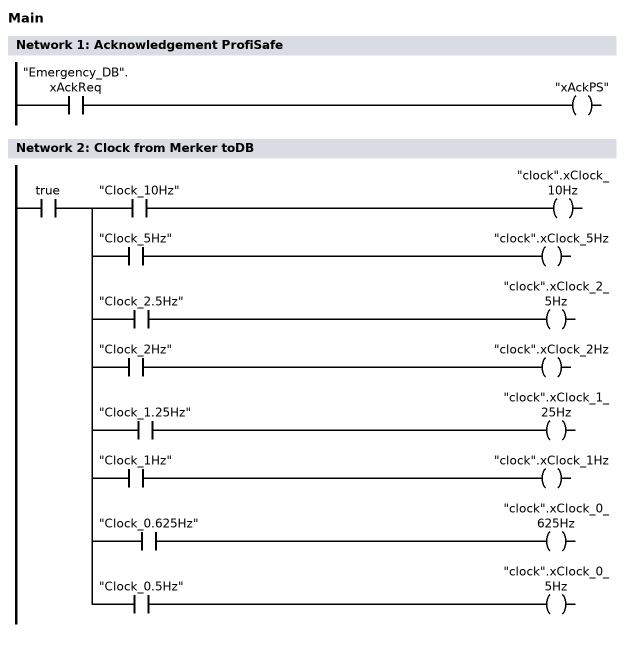
   RUNG wire#powerrail
      Contact( "Emergency_DB".xAckReq )
      Coil( "xAckPS" )
   END_RUNG
   // the same network as SCL:
   "xAckPS" := "Emergency_DB".xAckReq;
END_REGION

REGION Network 2: Clock from Merker toDB
   RUNG wire#powerrail
      Contact( true )
      wire#w1
      Contact( "Clock_10Hz" )
      Coil( "clock".xClock_10Hz )
   END_RUNG
   RUNG wire#w1
      Contact( "Clock_5Hz" )
      Coil( "clock".xClock_5Hz )
   END_RUNG
   RUNG wire#w1
      Contact( "Clock_2.5Hz" )
      Coil( "clock".xClock_2_5Hz )
   END_RUNG
   RUNG wire#w1
      Contact( "Clock_2Hz" )
      Coil( "clock".xClock_2Hz )
   END_RUNG
   RUNG wire#w1
      Contact( "Clock_1.25Hz" )
      Coil( "clock".xClock_1_25Hz )
   END_RUNG
   RUNG wire#w1
      Contact( "Clock_1Hz" )
      Coil( "clock".xClock_1Hz )
   END_RUNG
   RUNG wire#w1
      Contact( "Clock_0.625Hz" )
      Coil( "clock".xClock_0_625Hz )
   END_RUNG
   RUNG wire#w1
      Contact( "Clock_0.5Hz" )
      Coil( "clock".xClock_0_5Hz )
   END_RUNG
   // the same network as SCL:
   "clock".xClock_10Hz := true AND "Clock_10Hz";
   "clock".xClock_5Hz := true AND "Clock_5Hz";
   "clock".xClock_2_5Hz := true AND "Clock_2.5Hz";
   "clock".xClock_2Hz := true AND "Clock_2Hz";
   "clock".xClock_1_25Hz := true AND "Clock_1.25Hz";
   "clock".xClock_1Hz := true AND "Clock_1Hz";
   "clock".xClock_0_625Hz := true AND "Clock_0.625Hz";
   "clock".xClock_0_5Hz := true AND "Clock_0.5Hz";
END_REGION
END_ORGANIZATION_BLOCK

ORGANIZATION_BLOCK "Cyclic interrupt 100ms"   // OB33, LAD, CyclicInterrupt
{ S7_Optimized_Access := 'TRUE' }
VERSION : 0.1
// stored: AutoNumber false, IsIECCheckEnabled false, SetENOAutomatically false
   VAR_INPUT
      Initial_Call : Bool;   // Initial call of this OB
      Event_Count : Int;   // Events discarded
   END_VAR
BEGIN

REGION Network 1
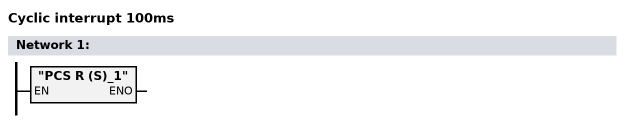
   RUNG wire#powerrail
      "PCS R (S)_1"()
   END_RUNG
   // the same network as SCL:
   "PCS R (S)_1"();
END_REGION
END_ORGANIZATION_BLOCK

FUNCTION "PCS R (S)_1" : Void   // FC46, LAD
TITLE = ModBus TCP for PCS Power Electronics
{ S7_Optimized_Access := 'TRUE' }
VERSION : 0.1
// stored: AutoNumber true, IsIECCheckEnabled false, SetENOAutomatically false, UDAEnableTagReadback false
   VAR_TEMP
      rVac : Real;
   END_VAR
   VAR_TEMP   // added for the SCL form of the ladder/FBD networks
      _w1 : Bool;
   END_VAR
BEGIN

REGION Network 1: Function Modbus Client
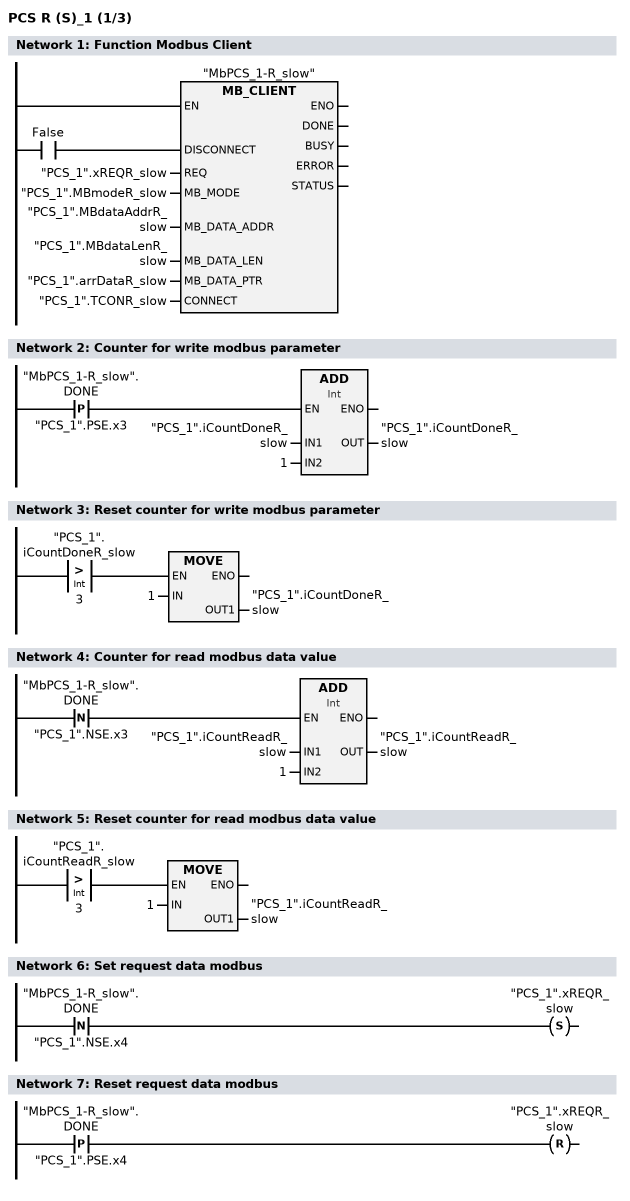
   RUNG wire#powerrail
      "MbPCS_1-R_slow".MB_CLIENT(DISCONNECT := wire#w1, REQ := "PCS_1".xREQR_slow, MB_MODE := "PCS_1".MBmodeR_slow, MB_DATA_ADDR := "PCS_1".MBdataAddrR_slow, MB_DATA_LEN := "PCS_1".MBdataLenR_slow, MB_DATA_PTR := "PCS_1".arrDataR_slow, CONNECT := "PCS_1".TCONR_slow, DONE =>, BUSY =>, ERROR =>, STATUS =>)
   END_RUNG
   RUNG wire#powerrail
      Contact( False )
   END_RUNG wire#w1
   // the same network as SCL:
   "MbPCS_1-R_slow"(DISCONNECT := False,   // MB_CLIENT
                    REQ := "PCS_1".xREQR_slow,
                    MB_MODE := "PCS_1".MBmodeR_slow,
                    MB_DATA_ADDR := "PCS_1".MBdataAddrR_slow,
                    MB_DATA_LEN := "PCS_1".MBdataLenR_slow,
                    MB_DATA_PTR := "PCS_1".arrDataR_slow,
                    CONNECT := "PCS_1".TCONR_slow);
END_REGION

REGION Network 2: Counter for write modbus parameter
   RUNG wire#powerrail
      P_Contact(operand := "MbPCS_1-R_slow".DONE, bit := "PCS_1".PSE.x3)
      { S7_Templates := "SrcType := Int" } Add(in1 := "PCS_1".iCountDoneR_slow, in2 := 1, out => "PCS_1".iCountDoneR_slow)
   END_RUNG
   // the same network as SCL:
   #_w1 := "MbPCS_1-R_slow".DONE AND NOT "PCS_1".PSE.x3;   // rising edge of "MbPCS_1-R_slow".DONE
   "PCS_1".PSE.x3 := "MbPCS_1-R_slow".DONE;
   IF #_w1 THEN "PCS_1".iCountDoneR_slow := "PCS_1".iCountDoneR_slow + 1; END_IF;
END_REGION

REGION Network 3: Reset counter for write modbus parameter
   RUNG wire#powerrail
      { S7_Templates := "SrcType := Int" } GT_Contact(in1 := "PCS_1".iCountDoneR_slow, in2 := 3)
      Move(in := 1, out1 => "PCS_1".iCountDoneR_slow)
   END_RUNG
   // the same network as SCL:
   IF "PCS_1".iCountDoneR_slow > 3 THEN "PCS_1".iCountDoneR_slow := 1; END_IF;
END_REGION

REGION Network 4: Counter for read modbus data value
   RUNG wire#powerrail
      N_Contact(operand := "MbPCS_1-R_slow".DONE, bit := "PCS_1".NSE.x3)
      { S7_Templates := "SrcType := Int" } Add(in1 := "PCS_1".iCountReadR_slow, in2 := 1, out => "PCS_1".iCountReadR_slow)
   END_RUNG
   // the same network as SCL:
   #_w1 := NOT "MbPCS_1-R_slow".DONE AND "PCS_1".NSE.x3;   // falling edge of "MbPCS_1-R_slow".DONE
   "PCS_1".NSE.x3 := "MbPCS_1-R_slow".DONE;
   IF #_w1 THEN "PCS_1".iCountReadR_slow := "PCS_1".iCountReadR_slow + 1; END_IF;
END_REGION

REGION Network 5: Reset counter for read modbus data value
   RUNG wire#powerrail
      { S7_Templates := "SrcType := Int" } GT_Contact(in1 := "PCS_1".iCountReadR_slow, in2 := 3)
      Move(in := 1, out1 => "PCS_1".iCountReadR_slow)
   END_RUNG
   // the same network as SCL:
   IF "PCS_1".iCountReadR_slow > 3 THEN "PCS_1".iCountReadR_slow := 1; END_IF;
END_REGION

REGION Network 6: Set request data modbus
   RUNG wire#powerrail
      N_Contact(operand := "MbPCS_1-R_slow".DONE, bit := "PCS_1".NSE.x4)
      S_Coil( "PCS_1".xREQR_slow )
   END_RUNG
   // the same network as SCL:
   #_w1 := NOT "MbPCS_1-R_slow".DONE AND "PCS_1".NSE.x4;   // falling edge of "MbPCS_1-R_slow".DONE
   "PCS_1".NSE.x4 := "MbPCS_1-R_slow".DONE;
   IF #_w1 THEN "PCS_1".xREQR_slow := TRUE; END_IF;
END_REGION

REGION Network 7: Reset request data modbus
   RUNG wire#powerrail
      P_Contact(operand := "MbPCS_1-R_slow".DONE, bit := "PCS_1".PSE.x4)
      R_Coil( "PCS_1".xREQR_slow )
   END_RUNG
   // the same network as SCL:
   #_w1 := "MbPCS_1-R_slow".DONE AND NOT "PCS_1".PSE.x4;   // rising edge of "MbPCS_1-R_slow".DONE
   "PCS_1".PSE.x4 := "MbPCS_1-R_slow".DONE;
   IF #_w1 THEN "PCS_1".xREQR_slow := FALSE; END_IF;
END_REGION

REGION Network 9: Write RW_Block1 parameter - da controllare password
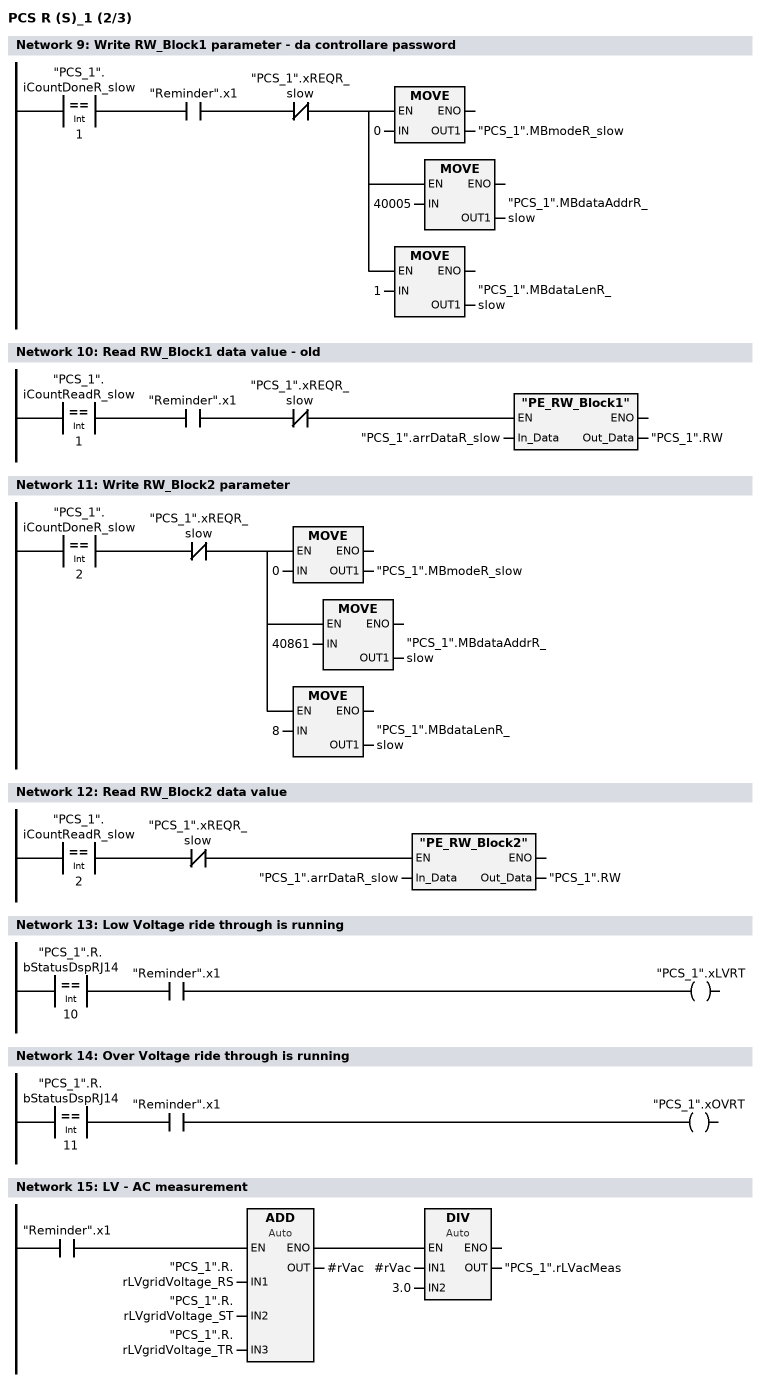
   RUNG wire#powerrail
      { S7_Templates := "SrcType := Int" } EQ_Contact(in1 := "PCS_1".iCountDoneR_slow, in2 := 1)
      Contact( "Reminder".x1 )
      I_Contact( "PCS_1".xREQR_slow )
      wire#w1
      Move(in := 0, out1 => "PCS_1".MBmodeR_slow)
   END_RUNG
   RUNG wire#w1
      Move(in := 40005, out1 => "PCS_1".MBdataAddrR_slow)
   END_RUNG
   RUNG wire#w1
      Move(in := 1, out1 => "PCS_1".MBdataLenR_slow)
   END_RUNG
   // the same network as SCL:
   IF ("PCS_1".iCountDoneR_slow = 1) AND "Reminder".x1 AND NOT "PCS_1".xREQR_slow THEN
       "PCS_1".MBmodeR_slow := 0;
       "PCS_1".MBdataAddrR_slow := 40005;
       "PCS_1".MBdataLenR_slow := 1;
   END_IF;
END_REGION

REGION Network 10: Read RW_Block1 data value - old
   RUNG wire#powerrail
      { S7_Templates := "SrcType := Int" } EQ_Contact(in1 := "PCS_1".iCountReadR_slow, in2 := 1)
      Contact( "Reminder".x1 )
      I_Contact( "PCS_1".xREQR_slow )
      "PE_RW_Block1"(In_Data := "PCS_1".arrDataR_slow, Out_Data => "PCS_1".RW)
   END_RUNG
   // the same network as SCL:
   IF ("PCS_1".iCountReadR_slow = 1) AND "Reminder".x1 AND NOT "PCS_1".xREQR_slow THEN
       "PE_RW_Block1"(In_Data := "PCS_1".arrDataR_slow, Out_Data => "PCS_1".RW);
   END_IF;
END_REGION

REGION Network 11: Write RW_Block2 parameter
   RUNG wire#powerrail
      { S7_Templates := "SrcType := Int" } EQ_Contact(in1 := "PCS_1".iCountDoneR_slow, in2 := 2)
      I_Contact( "PCS_1".xREQR_slow )
      wire#w1
      Move(in := 0, out1 => "PCS_1".MBmodeR_slow)
   END_RUNG
   RUNG wire#w1
      Move(in := 40861, out1 => "PCS_1".MBdataAddrR_slow)
   END_RUNG
   RUNG wire#w1
      Move(in := 8, out1 => "PCS_1".MBdataLenR_slow)
   END_RUNG
   // the same network as SCL:
   IF ("PCS_1".iCountDoneR_slow = 2) AND NOT "PCS_1".xREQR_slow THEN
       "PCS_1".MBmodeR_slow := 0;
       "PCS_1".MBdataAddrR_slow := 40861;
       "PCS_1".MBdataLenR_slow := 8;
   END_IF;
END_REGION

REGION Network 12: Read RW_Block2 data value
   RUNG wire#powerrail
      { S7_Templates := "SrcType := Int" } EQ_Contact(in1 := "PCS_1".iCountReadR_slow, in2 := 2)
      I_Contact( "PCS_1".xREQR_slow )
      "PE_RW_Block2"(In_Data := "PCS_1".arrDataR_slow, Out_Data => "PCS_1".RW)
   END_RUNG
   // the same network as SCL:
   IF ("PCS_1".iCountReadR_slow = 2) AND NOT "PCS_1".xREQR_slow THEN
       "PE_RW_Block2"(In_Data := "PCS_1".arrDataR_slow, Out_Data => "PCS_1".RW);
   END_IF;
END_REGION

REGION Network 13: Low Voltage ride through is running
   RUNG wire#powerrail
      { S7_Templates := "SrcType := Int" } EQ_Contact(in1 := "PCS_1".R.bStatusDspRJ14, in2 := 10)
      Contact( "Reminder".x1 )
      Coil( "PCS_1".xLVRT )
   END_RUNG
   // the same network as SCL:
   "PCS_1".xLVRT := ("PCS_1".R.bStatusDspRJ14 = 10) AND "Reminder".x1;
END_REGION

REGION Network 14: Over Voltage ride through is running
   RUNG wire#powerrail
      { S7_Templates := "SrcType := Int" } EQ_Contact(in1 := "PCS_1".R.bStatusDspRJ14, in2 := 11)
      Contact( "Reminder".x1 )
      Coil( "PCS_1".xOVRT )
   END_RUNG
   // the same network as SCL:
   "PCS_1".xOVRT := ("PCS_1".R.bStatusDspRJ14 = 11) AND "Reminder".x1;
END_REGION

REGION Network 15: LV - AC measurement
   RUNG wire#powerrail
      Contact( "Reminder".x1 )
      Add(in1 := "PCS_1".R.rLVgridVoltage_RS, in2 := "PCS_1".R.rLVgridVoltage_ST, in3 := "PCS_1".R.rLVgridVoltage_TR, out => #rVac)
      Div(in1 := #rVac, in2 := 3.0, out => "PCS_1".rLVacMeas)
   END_RUNG
   // the same network as SCL:
   IF "Reminder".x1 THEN
       #rVac := "PCS_1".R.rLVgridVoltage_RS + "PCS_1".R.rLVgridVoltage_ST + "PCS_1".R.rLVgridVoltage_TR;
       "PCS_1".rLVacMeas := #rVac / 3.0;
   END_IF;
END_REGION

REGION Network 16: MV - AC measurement
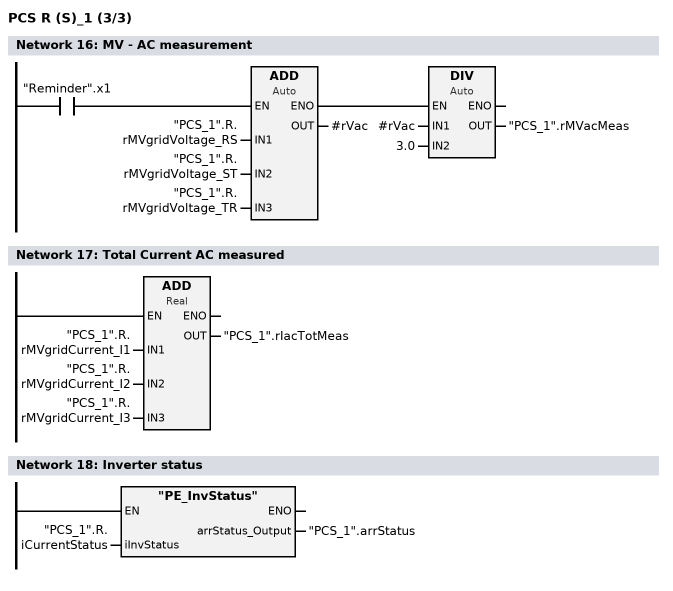
   RUNG wire#powerrail
      Contact( "Reminder".x1 )
      Add(in1 := "PCS_1".R.rMVgridVoltage_RS, in2 := "PCS_1".R.rMVgridVoltage_ST, in3 := "PCS_1".R.rMVgridVoltage_TR, out => #rVac)
      Div(in1 := #rVac, in2 := 3.0, out => "PCS_1".rMVacMeas)
   END_RUNG
   // the same network as SCL:
   IF "Reminder".x1 THEN
       #rVac := "PCS_1".R.rMVgridVoltage_RS + "PCS_1".R.rMVgridVoltage_ST + "PCS_1".R.rMVgridVoltage_TR;
       "PCS_1".rMVacMeas := #rVac / 3.0;
   END_IF;
END_REGION

REGION Network 17: Total Current AC measured
   RUNG wire#powerrail
      { S7_Templates := "SrcType := Real" } Add(in1 := "PCS_1".R.rMVgridCurrent_I1, in2 := "PCS_1".R.rMVgridCurrent_I2, in3 := "PCS_1".R.rMVgridCurrent_I3, out => "PCS_1".rIacTotMeas)
   END_RUNG
   // the same network as SCL:
   "PCS_1".rIacTotMeas := "PCS_1".R.rMVgridCurrent_I1 + "PCS_1".R.rMVgridCurrent_I2 + "PCS_1".R.rMVgridCurrent_I3;
END_REGION

REGION Network 18: Inverter status
   RUNG wire#powerrail
      "PE_InvStatus"(iInvStatus := "PCS_1".R.iCurrentStatus, arrStatus_Output => "PCS_1".arrStatus)
   END_RUNG
   // the same network as SCL:
   "PE_InvStatus"(iInvStatus := "PCS_1".R.iCurrentStatus, arrStatus_Output => "PCS_1".arrStatus);
END_REGION
END_FUNCTION

FUNCTION "PE_RW_Block1" : Void
{ S7_Optimized_Access := 'TRUE' }
VERSION : 0.1
   VAR_INPUT 
      In_Data : Array[1..125] of Word;   // pcs
   END_VAR

   VAR_OUTPUT 
      Out_Data : "RW_PE";
   END_VAR


BEGIN
	REGION
	    // 2022/01/24
	END_REGION
	
	REGION
	    
	    #Out_Data.iUserPswIns := WORD_TO_INT(#In_Data[1]);
	    
	END_REGION
END_FUNCTION

FUNCTION "PE_RW_Block2" : Void
{ S7_Optimized_Access := 'TRUE' }
VERSION : 0.1
   VAR_INPUT 
      In_Data : Array[1..125] of Word;   // pcs
   END_VAR

   VAR_OUTPUT 
      Out_Data : "RW_PE";
   END_VAR


BEGIN
	//27-03-2023
	
	REGION
	    
	    #Out_Data.iModePctrlCmd := WORD_TO_INT(#In_Data[1]);
	    #Out_Data.iModeQctrlCmd := WORD_TO_INT(#In_Data[2]);
	    #Out_Data.rPacRef       := INT_TO_REAL(WORD_TO_INT(#In_Data[3]))/100.0;
	    #Out_Data.rQacRef       := INT_TO_REAL(WORD_TO_INT(#In_Data[8]))/100.0;
	    
	END_REGION
END_FUNCTION

FUNCTION "PE_InvStatus" : Void
{ S7_Optimized_Access := 'TRUE' }
VERSION : 0.1
   VAR_INPUT 
      iInvStatus : Int;   // Signal coming from Modbus read
   END_VAR

   VAR_OUTPUT 
      arrStatus_Output : Array[0..17] of Bool;
   END_VAR

   VAR_TEMP 
      arrStatus : Array[0..17] of Bool;
      i : Int;
   END_VAR


BEGIN
	CASE #iInvStatus OF
	    0:
	        #arrStatus[0] := TRUE;
	    1:
	        #arrStatus[1] := TRUE;
	    2:
	        #arrStatus[2] := TRUE;
	    3:
	        #arrStatus[3] := TRUE;
	    4:
	        #arrStatus[4] := TRUE;
	    5:
	        #arrStatus[5] := TRUE;
	    6:
	        #arrStatus[6] := TRUE;
	    7:
	        #arrStatus[7] := TRUE;
	    8:
	        #arrStatus[8] := TRUE;
	    9:
	        #arrStatus[9] := TRUE;
	    10:
	        #arrStatus[10] := TRUE;
	    11:
	        #arrStatus[11] := TRUE;
	    12:
	        #arrStatus[12] := TRUE;
	    13:
	        #arrStatus[13] := TRUE;
	    14:
	        #arrStatus[14] := TRUE;
	    15:
	        #arrStatus[15] := TRUE;
	    16:
	        #arrStatus[16] := TRUE;
	    17:
	        #arrStatus[17] := TRUE;
	    ELSE
	        FOR #i := 0 TO 17 DO                //if number out of range full array to zero
	            #arrStatus [#i]:= FALSE;
	        END_FOR;
	END_CASE;
	
	#arrStatus_Output := #arrStatus;    //copy of local array
	
	
	
END_FUNCTION

ORGANIZATION_BLOCK "Cyclic interrupt 1s"   // OB35, LAD, CyclicInterrupt
{ S7_Optimized_Access := 'TRUE' }
VERSION : 0.1
// stored: AutoNumber false, IsIECCheckEnabled false, SetENOAutomatically false
   VAR_INPUT
      Initial_Call : Bool;   // Initial call of this OB
      Event_Count : Int;   // Events discarded
   END_VAR
BEGIN

REGION Network 1: Heartbeat BMS1
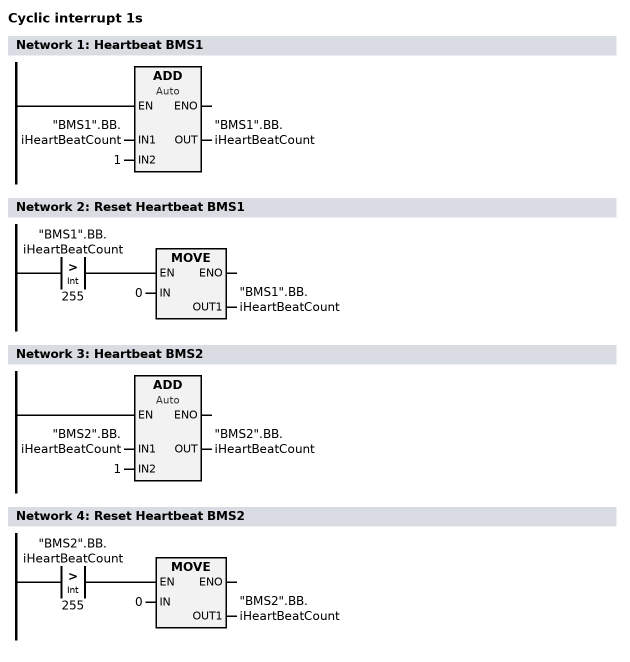
   RUNG wire#powerrail
      Add(in1 := "BMS1".BB.iHeartBeatCount, in2 := 1, out => "BMS1".BB.iHeartBeatCount)
   END_RUNG
   // the same network as SCL:
   "BMS1".BB.iHeartBeatCount := "BMS1".BB.iHeartBeatCount + 1;
END_REGION

REGION Network 2: Reset Heartbeat BMS1
   RUNG wire#powerrail
      { S7_Templates := "SrcType := Int" } GT_Contact(in1 := "BMS1".BB.iHeartBeatCount, in2 := 255)
      Move(in := 0, out1 => "BMS1".BB.iHeartBeatCount)
   END_RUNG
   // the same network as SCL:
   IF "BMS1".BB.iHeartBeatCount > 255 THEN "BMS1".BB.iHeartBeatCount := 0; END_IF;
END_REGION

REGION Network 3: Heartbeat BMS2
   RUNG wire#powerrail
      Add(in1 := "BMS2".BB.iHeartBeatCount, in2 := 1, out => "BMS2".BB.iHeartBeatCount)
   END_RUNG
   // the same network as SCL:
   "BMS2".BB.iHeartBeatCount := "BMS2".BB.iHeartBeatCount + 1;
END_REGION

REGION Network 4: Reset Heartbeat BMS2
   RUNG wire#powerrail
      { S7_Templates := "SrcType := Int" } GT_Contact(in1 := "BMS2".BB.iHeartBeatCount, in2 := 255)
      Move(in := 0, out1 => "BMS2".BB.iHeartBeatCount)
   END_RUNG
   // the same network as SCL:
   IF "BMS2".BB.iHeartBeatCount > 255 THEN "BMS2".BB.iHeartBeatCount := 0; END_IF;
END_REGION
END_ORGANIZATION_BLOCK

ORGANIZATION_BLOCK "Cyclic interrupt 20ms"   // OB31, LAD, CyclicInterrupt
{ S7_Optimized_Access := 'TRUE' }
VERSION : 0.1
// stored: AutoNumber false, IsIECCheckEnabled false, SetENOAutomatically false
   VAR_INPUT
      Initial_Call : Bool;   // Initial call of this OB
      Event_Count : Int;   // Events discarded
   END_VAR
BEGIN
END_ORGANIZATION_BLOCK

ORGANIZATION_BLOCK "Cyclic interrupt 500ms"   // OB34, LAD, CyclicInterrupt
{ S7_Optimized_Access := 'TRUE' }
VERSION : 0.1
// stored: AutoNumber false, IsIECCheckEnabled false, SetENOAutomatically false
   VAR_INPUT
      Initial_Call : Bool;   // Initial call of this OB
      Event_Count : Int;   // Events discarded
   END_VAR
BEGIN
END_ORGANIZATION_BLOCK

ORGANIZATION_BLOCK "Cyclic interrupt 50ms"   // OB32, LAD, CyclicInterrupt
{ S7_Optimized_Access := 'TRUE' }
VERSION : 0.1
// stored: AutoNumber true, IsIECCheckEnabled false, SetENOAutomatically false
   VAR_INPUT
      Initial_Call : Bool;   // Initial call of this OB
      Event_Count : Int;   // Events discarded
   END_VAR
BEGIN
END_ORGANIZATION_BLOCK

ORGANIZATION_BLOCK "ProfiNet 10ms"   // OB30, LAD, CyclicInterrupt
{ S7_Optimized_Access := 'TRUE' }
VERSION : 0.1
// stored: AutoNumber true, IsIECCheckEnabled false, SetENOAutomatically false
   VAR_INPUT
      Initial_Call : Bool;   // Initial call of this OB
      Event_Count : Int;   // Events discarded
   END_VAR
   VAR_TEMP
      Ret_val : Int;
   END_VAR
BEGIN

REGION Network 1: Diagnostic Profinet Module (CPU is Module 1)
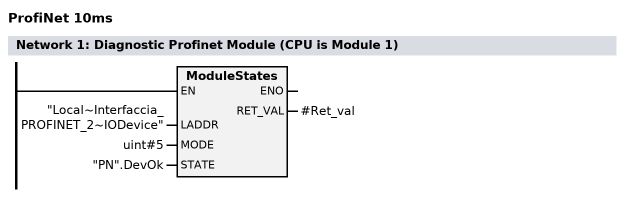
   RUNG wire#powerrail
      ModuleStates(LADDR := "Local~Interfaccia_PROFINET_2~IODevice", MODE := uint#5, STATE := "PN".DevOk, Ret_Val => #Ret_val)
   END_RUNG
   // the same network as SCL:
   #Ret_val := ModuleStates(LADDR := "Local~Interfaccia_PROFINET_2~IODevice",
                           MODE := uint#5,
                           STATE := "PN".DevOk);
END_REGION
END_ORGANIZATION_BLOCK

ORGANIZATION_BLOCK "Startup"   // OB124, LAD, Startup
TITLE = "Complete Restart"
{ S7_Optimized_Access := 'TRUE' }
VERSION : 0.1
// stored: AutoNumber true, IsIECCheckEnabled false, SetENOAutomatically false
   VAR_INPUT
      LostRetentive : Bool;   // True if retentive data are lost
      LostRTC : Bool;   // True if date and time are lost
   END_VAR
BEGIN

REGION Network 1
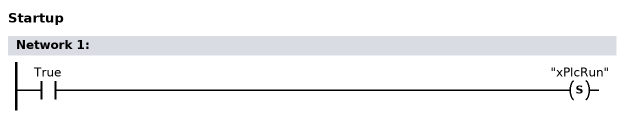
   RUNG wire#powerrail
      Contact( True )
      S_Coil( "xPlcRun" )
   END_RUNG
   // the same network as SCL:
   IF True THEN "xPlcRun" := TRUE; END_IF;
END_REGION
END_ORGANIZATION_BLOCK

FUNCTION "test_2" : Void   // FC4, LAD
{ S7_Optimized_Access := 'TRUE' }
VERSION : 0.1
// stored: AutoNumber true, IsIECCheckEnabled false, SetENOAutomatically false, UDAEnableTagReadback false
   VAR_TEMP
      ixT1 : S5Time;
   END_VAR
BEGIN
END_FUNCTION

FUNCTION "SS Alarms" : Void   // FC102, LAD
{ S7_Optimized_Access := 'TRUE' }
VERSION : 0.1
// stored: AutoNumber false, IsIECCheckEnabled false, SetENOAutomatically false, UDAEnableTagReadback false
BEGIN

REGION Network 1: Alarm Status On/Off
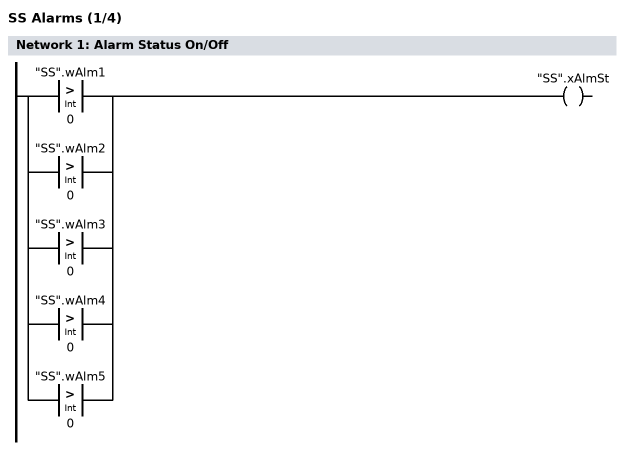
   RUNG wire#powerrail
      { S7_Templates := "SrcType := Int" } GT_Contact(in1 := "SS".wAlm1, in2 := 0)
      wire#w1
      Coil( "SS".xAlmSt )
   END_RUNG
   RUNG wire#powerrail
      { S7_Templates := "SrcType := Int" } GT_Contact(in1 := "SS".wAlm2, in2 := 0)
   END_RUNG wire#w1
   RUNG wire#powerrail
      { S7_Templates := "SrcType := Int" } GT_Contact(in1 := "SS".wAlm3, in2 := 0)
   END_RUNG wire#w1
   RUNG wire#powerrail
      { S7_Templates := "SrcType := Int" } GT_Contact(in1 := "SS".wAlm4, in2 := 0)
   END_RUNG wire#w1
   RUNG wire#powerrail
      { S7_Templates := "SrcType := Int" } GT_Contact(in1 := "SS".wAlm5, in2 := 0)
   END_RUNG wire#w1
   // the same network as SCL:
   "SS".xAlmSt := ("SS".wAlm1 > 0) OR ("SS".wAlm2 > 0) OR ("SS".wAlm3 > 0) OR ("SS".wAlm4 > 0) OR ("SS".wAlm5 > 0);
END_REGION

REGION Network 2: Alarm Word 1
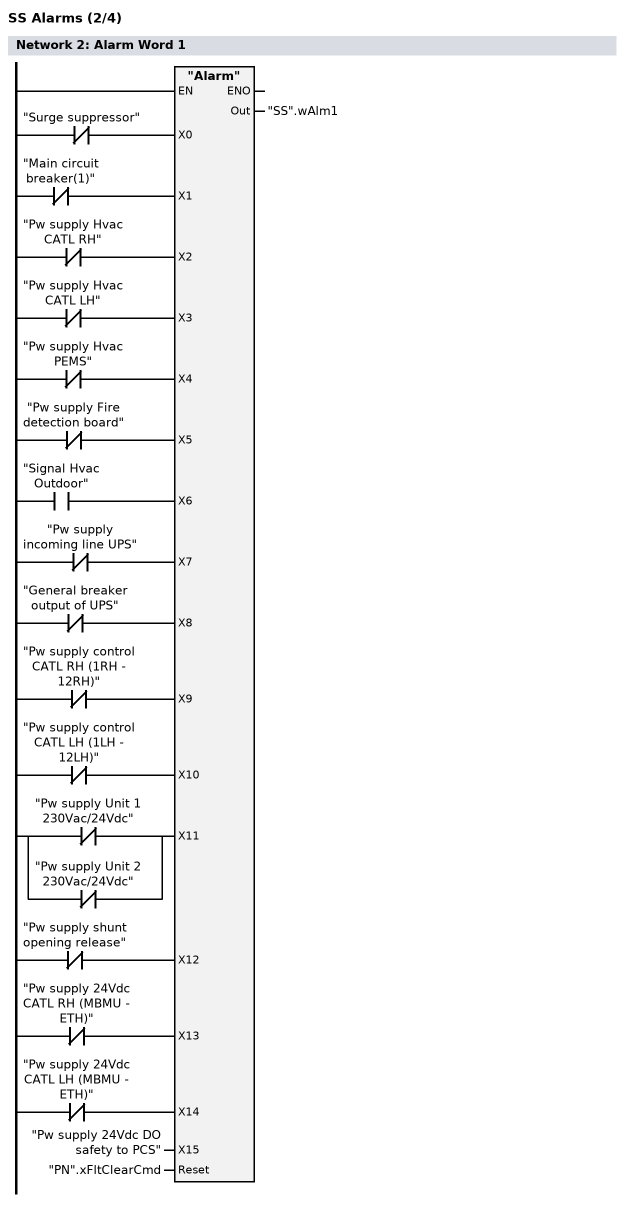
   RUNG wire#powerrail
      "Alarm"(X0 := wire#w1, X1 := wire#w2, X2 := wire#w3, X3 := wire#w4, X4 := wire#w5, X5 := wire#w6, X6 := wire#w7, X7 := wire#w8, X8 := wire#w9, X9 := wire#w10, X10 := wire#w11, X11 := wire#w12, X12 := wire#w13, X13 := wire#w14, X14 := wire#w15, X15 := "Pw supply 24Vdc DO safety to PCS", Reset := "PN".xFltClearCmd, Out => "SS".wAlm1)
   END_RUNG
   RUNG wire#powerrail
      I_Contact( "Surge suppressor" )
   END_RUNG wire#w1
   RUNG wire#powerrail
      I_Contact( "Main circuit breaker(1)" )
   END_RUNG wire#w2
   RUNG wire#powerrail
      I_Contact( "Pw supply Hvac CATL RH" )
   END_RUNG wire#w3
   RUNG wire#powerrail
      I_Contact( "Pw supply Hvac CATL LH" )
   END_RUNG wire#w4
   RUNG wire#powerrail
      I_Contact( "Pw supply Hvac PEMS" )
   END_RUNG wire#w5
   RUNG wire#powerrail
      I_Contact( "Pw supply Fire detection board" )
   END_RUNG wire#w6
   RUNG wire#powerrail
      Contact( "Signal Hvac Outdoor" )
   END_RUNG wire#w7
   RUNG wire#powerrail
      I_Contact( "Pw supply incoming line UPS" )
   END_RUNG wire#w8
   RUNG wire#powerrail
      I_Contact( "General breaker output of UPS" )
   END_RUNG wire#w9
   RUNG wire#powerrail
      I_Contact( "Pw supply control CATL RH (1RH - 12RH)" )
   END_RUNG wire#w10
   RUNG wire#powerrail
      I_Contact( "Pw supply control CATL LH (1LH - 12LH)" )
   END_RUNG wire#w11
   RUNG wire#powerrail
      I_Contact( "Pw supply Unit 1 230Vac/24Vdc" )
   END_RUNG wire#w12
   RUNG wire#powerrail
      I_Contact( "Pw supply Unit 2 230Vac/24Vdc" )
   END_RUNG wire#w12
   RUNG wire#powerrail
      I_Contact( "Pw supply shunt opening release" )
   END_RUNG wire#w13
   RUNG wire#powerrail
      I_Contact( "Pw supply 24Vdc CATL RH (MBMU - ETH)" )
   END_RUNG wire#w14
   RUNG wire#powerrail
      I_Contact( "Pw supply 24Vdc CATL LH (MBMU - ETH)" )
   END_RUNG wire#w15
   // the same network as SCL:
   "Alarm"(X0 := NOT "Surge suppressor",
           X1 := NOT "Main circuit breaker(1)",
           X2 := NOT "Pw supply Hvac CATL RH",
           X3 := NOT "Pw supply Hvac CATL LH",
           X4 := NOT "Pw supply Hvac PEMS",
           X5 := NOT "Pw supply Fire detection board",
           X6 := "Signal Hvac Outdoor",
           X7 := NOT "Pw supply incoming line UPS",
           X8 := NOT "General breaker output of UPS",
           X9 := NOT "Pw supply control CATL RH (1RH - 12RH)",
           X10 := NOT "Pw supply control CATL LH (1LH - 12LH)",
           X11 := NOT "Pw supply Unit 1 230Vac/24Vdc" OR NOT "Pw supply Unit 2 230Vac/24Vdc",
           X12 := NOT "Pw supply shunt opening release",
           X13 := NOT "Pw supply 24Vdc CATL RH (MBMU - ETH)",
           X14 := NOT "Pw supply 24Vdc CATL LH (MBMU - ETH)",
           X15 := "Pw supply 24Vdc DO safety to PCS",
           Reset := "PN".xFltClearCmd,
           Out => "SS".wAlm1);
END_REGION

REGION Network 3: Alarm Word 2
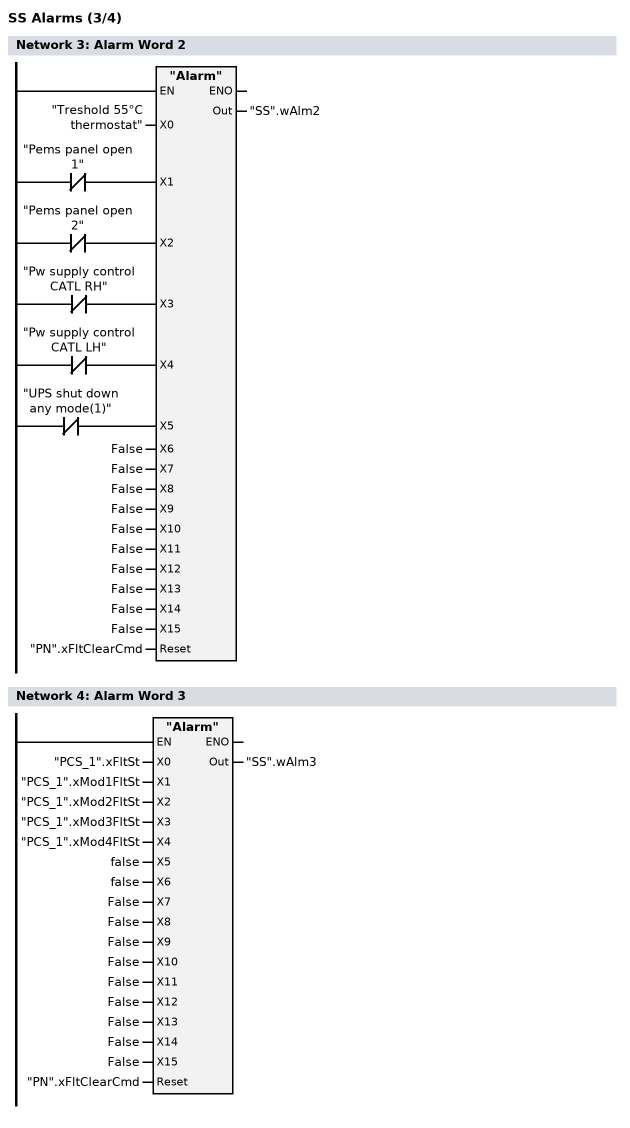
   RUNG wire#powerrail
      "Alarm"(X1 := wire#w1, X2 := wire#w2, X3 := wire#w3, X4 := wire#w4, X5 := wire#w5, X0 := "Treshold 55°C thermostat", X6 := False, X7 := False, X8 := False, X9 := False, X10 := False, X11 := False, X12 := False, X13 := False, X14 := False, X15 := False, Reset := "PN".xFltClearCmd, Out => "SS".wAlm2)
   END_RUNG
   RUNG wire#powerrail
      I_Contact( "Pems panel open 1" )
   END_RUNG wire#w1
   RUNG wire#powerrail
      I_Contact( "Pems panel open 2" )
   END_RUNG wire#w2
   RUNG wire#powerrail
      I_Contact( "Pw supply control CATL RH" )
   END_RUNG wire#w3
   RUNG wire#powerrail
      I_Contact( "Pw supply control CATL LH" )
   END_RUNG wire#w4
   RUNG wire#powerrail
      I_Contact( "UPS shut down any mode(1)" )
   END_RUNG wire#w5
   // the same network as SCL:
   "Alarm"(X0 := "Treshold 55°C thermostat",
           X1 := NOT "Pems panel open 1",
           X2 := NOT "Pems panel open 2",
           X3 := NOT "Pw supply control CATL RH",
           X4 := NOT "Pw supply control CATL LH",
           X5 := NOT "UPS shut down any mode(1)",
           X6 := False,
           X7 := False,
           X8 := False,
           X9 := False,
           X10 := False,
           X11 := False,
           X12 := False,
           X13 := False,
           X14 := False,
           X15 := False,
           Reset := "PN".xFltClearCmd,
           Out => "SS".wAlm2);
END_REGION

REGION Network 4: Alarm Word 3
   RUNG wire#powerrail
      "Alarm"(X0 := "PCS_1".xFltSt, X1 := "PCS_1".xMod1FltSt, X2 := "PCS_1".xMod2FltSt, X3 := "PCS_1".xMod3FltSt, X4 := "PCS_1".xMod4FltSt, X5 := false, X6 := false, X7 := False, X8 := False, X9 := False, X10 := False, X11 := False, X12 := False, X13 := False, X14 := False, X15 := False, Reset := "PN".xFltClearCmd, Out => "SS".wAlm3)
   END_RUNG
   // the same network as SCL:
   "Alarm"(X0 := "PCS_1".xFltSt,
           X1 := "PCS_1".xMod1FltSt,
           X2 := "PCS_1".xMod2FltSt,
           X3 := "PCS_1".xMod3FltSt,
           X4 := "PCS_1".xMod4FltSt,
           X5 := false,
           X6 := false,
           X7 := False,
           X8 := False,
           X9 := False,
           X10 := False,
           X11 := False,
           X12 := False,
           X13 := False,
           X14 := False,
           X15 := False,
           Reset := "PN".xFltClearCmd,
           Out => "SS".wAlm3);
END_REGION

REGION Network 5: Alarm Word 4
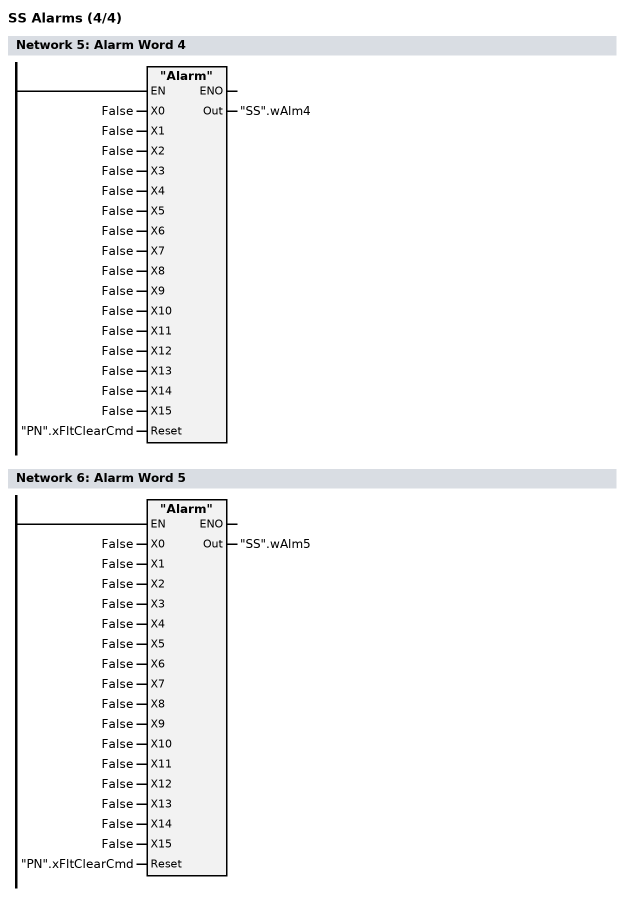
   RUNG wire#powerrail
      "Alarm"(X0 := False, X1 := False, X2 := False, X3 := False, X4 := False, X5 := False, X6 := False, X7 := False, X8 := False, X9 := False, X10 := False, X11 := False, X12 := False, X13 := False, X14 := False, X15 := False, Reset := "PN".xFltClearCmd, Out => "SS".wAlm4)
   END_RUNG
   // the same network as SCL:
   "Alarm"(X0 := False,
           X1 := False,
           X2 := False,
           X3 := False,
           X4 := False,
           X5 := False,
           X6 := False,
           X7 := False,
           X8 := False,
           X9 := False,
           X10 := False,
           X11 := False,
           X12 := False,
           X13 := False,
           X14 := False,
           X15 := False,
           Reset := "PN".xFltClearCmd,
           Out => "SS".wAlm4);
END_REGION

REGION Network 6: Alarm Word 5
   RUNG wire#powerrail
      "Alarm"(X0 := False, X1 := False, X2 := False, X3 := False, X4 := False, X5 := False, X6 := False, X7 := False, X8 := False, X9 := False, X10 := False, X11 := False, X12 := False, X13 := False, X14 := False, X15 := False, Reset := "PN".xFltClearCmd, Out => "SS".wAlm5)
   END_RUNG
   // the same network as SCL:
   "Alarm"(X0 := False,
           X1 := False,
           X2 := False,
           X3 := False,
           X4 := False,
           X5 := False,
           X6 := False,
           X7 := False,
           X8 := False,
           X9 := False,
           X10 := False,
           X11 := False,
           X12 := False,
           X13 := False,
           X14 := False,
           X15 := False,
           Reset := "PN".xFltClearCmd,
           Out => "SS".wAlm5);
END_REGION
END_FUNCTION

FUNCTION "Alarm" : Void
{ S7_Optimized_Access := 'TRUE' }
VERSION : 0.1
   VAR_INPUT 
      X0 : Bool;
      X1 : Bool;
      X2 : Bool;
      X3 : Bool;
      X4 : Bool;
      X5 : Bool;
      X6 : Bool;
      X7 : Bool;
      X8 : Bool;
      X9 : Bool;
      X10 : Bool;
      X11 : Bool;
      X12 : Bool;
      X13 : Bool;
      X14 : Bool;
      X15 : Bool;
      Reset : Bool;
   END_VAR

   VAR_OUTPUT 
      Out : Word;
   END_VAR


BEGIN
	
	IF #X0
	    THEN
	    #Out.%X0 := True;
	END_IF;
	
	IF #X1
	THEN
	    #Out.%X1 := True;
	END_IF;
	
	IF #X2
	THEN
	    #Out.%X2 := True;
	END_IF;
	
	IF #X3
	THEN
	    #Out.%X3 := True;
	END_IF;
	
	IF #X4
	THEN
	    #Out.%X4 := True;
	END_IF;
	
	IF #X5
	THEN
	    #Out.%X5 := True;
	END_IF;
	
	IF #X6
	THEN
	    #Out.%X6 := True;
	END_IF;
	
	IF #X7
	THEN
	    #Out.%X7 := True;
	END_IF;
	
	IF #X8
	THEN
	    #Out.%X8 := True;
	END_IF;
	
	IF #X9
	THEN
	    #Out.%X9 := True;
	END_IF;
	
	IF #X10
	THEN
	    #Out.%X10 := True;
	END_IF;
	
	IF #X11
	THEN
	    #Out.%X11 := True;
	END_IF;
	
	IF #X12
	THEN
	    #Out.%X12 := True;
	END_IF;
	
	IF #X13
	THEN
	    #Out.%X13 := True;
	END_IF;
	
	IF #X14
	THEN
	    #Out.%X14 := True;
	END_IF;
	
	IF #X15
	THEN
	    #Out.%X15 := True;
	END_IF;
	
	IF #Reset
	THEN
	    #Out := 0;
	END_IF;
	
END_FUNCTION

FUNCTION "SS Faults" : Void   // FC101, LAD
{ S7_Optimized_Access := 'TRUE' }
VERSION : 0.1
// stored: AutoNumber false, IsIECCheckEnabled false, SetENOAutomatically false, UDAEnableTagReadback false
BEGIN

REGION Network 1: Fault Power Island
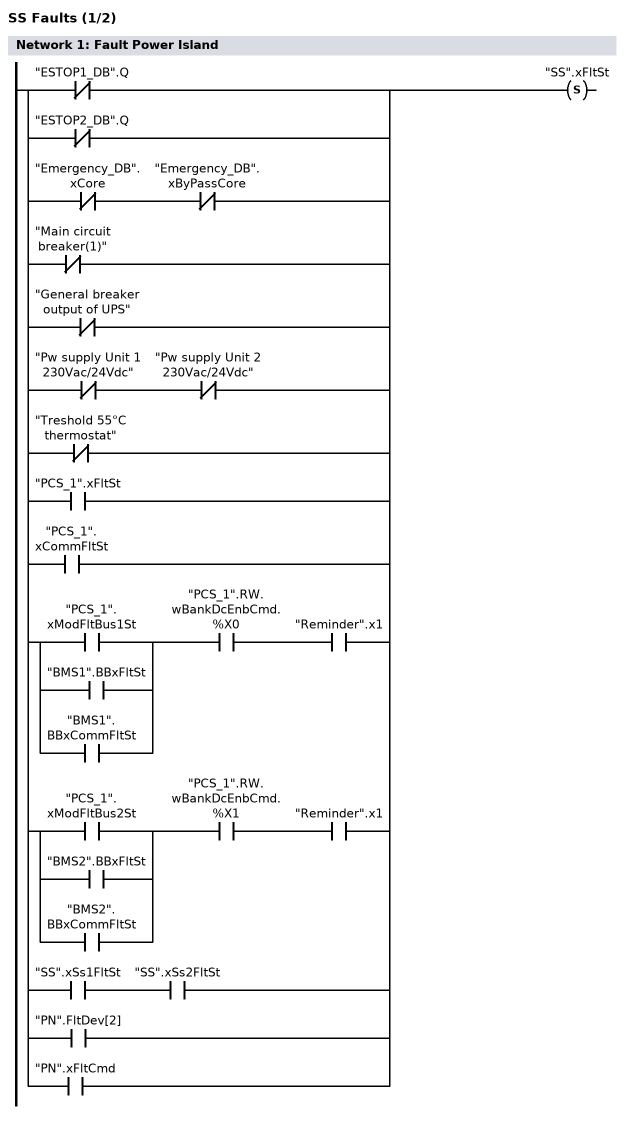
   RUNG wire#powerrail
      I_Contact( "ESTOP1_DB".Q )
      wire#w1
      S_Coil( "SS".xFltSt )
   END_RUNG
   RUNG wire#powerrail
      I_Contact( "ESTOP2_DB".Q )
   END_RUNG wire#w1
   RUNG wire#powerrail
      I_Contact( "Emergency_DB".xCore )
      I_Contact( "Emergency_DB".xByPassCore )
   END_RUNG wire#w1
   RUNG wire#powerrail
      I_Contact( "Main circuit breaker(1)" )
   END_RUNG wire#w1
   RUNG wire#powerrail
      I_Contact( "General breaker output of UPS" )
   END_RUNG wire#w1
   RUNG wire#powerrail
      I_Contact( "Pw supply Unit 1 230Vac/24Vdc" )
      I_Contact( "Pw supply Unit 2 230Vac/24Vdc" )
   END_RUNG wire#w1
   RUNG wire#powerrail
      I_Contact( "Treshold 55°C thermostat" )
   END_RUNG wire#w1
   RUNG wire#powerrail
      Contact( "PCS_1".xFltSt )
   END_RUNG wire#w1
   RUNG wire#powerrail
      Contact( "PCS_1".xCommFltSt )
   END_RUNG wire#w1
   RUNG wire#powerrail
      Contact( "PCS_1".xModFltBus1St )
      wire#w2
      Contact( "PCS_1".RW.wBankDcEnbCmd.%X0 )
      Contact( "Reminder".x1 )
   END_RUNG wire#w1
   RUNG wire#powerrail
      Contact( "BMS1".BBxFltSt )
   END_RUNG wire#w2
   RUNG wire#powerrail
      Contact( "BMS1".BBxCommFltSt )
   END_RUNG wire#w2
   RUNG wire#powerrail
      Contact( "PCS_1".xModFltBus2St )
      wire#w3
      Contact( "PCS_1".RW.wBankDcEnbCmd.%X1 )
      Contact( "Reminder".x1 )
   END_RUNG wire#w1
   RUNG wire#powerrail
      Contact( "BMS2".BBxFltSt )
   END_RUNG wire#w3
   RUNG wire#powerrail
      Contact( "BMS2".BBxCommFltSt )
   END_RUNG wire#w3
   RUNG wire#powerrail
      Contact( "SS".xSs1FltSt )
      Contact( "SS".xSs2FltSt )
   END_RUNG wire#w1
   RUNG wire#powerrail
      Contact( "PN".FltDev[2] )
   END_RUNG wire#w1
   RUNG wire#powerrail
      Contact( "PN".xFltCmd )
   END_RUNG wire#w1
   // the same network as SCL:
   IF NOT "ESTOP1_DB".Q OR NOT "ESTOP2_DB".Q OR (NOT "Emergency_DB".xCore AND NOT "Emergency_DB".xByPassCore) OR NOT "Main circuit breaker(1)" OR NOT "General breaker output of UPS" OR (NOT "Pw supply Unit 1 230Vac/24Vdc" AND NOT "Pw supply Unit 2 230Vac/24Vdc") OR NOT "Treshold 55°C thermostat" OR "PCS_1".xFltSt OR "PCS_1".xCommFltSt OR (("PCS_1".xModFltBus1St OR "BMS1".BBxFltSt OR "BMS1".BBxCommFltSt) AND "PCS_1".RW.wBankDcEnbCmd.%X0 AND "Reminder".x1) OR (("PCS_1".xModFltBus2St OR "BMS2".BBxFltSt OR "BMS2".BBxCommFltSt) AND "PCS_1".RW.wBankDcEnbCmd.%X1 AND "Reminder".x1) OR ("SS".xSs1FltSt AND "SS".xSs2FltSt) OR "PN".FltDev[2] OR "PN".xFltCmd THEN
       "SS".xFltSt := TRUE;
   END_IF;
END_REGION

REGION Network 2: Fault Subsystem 1
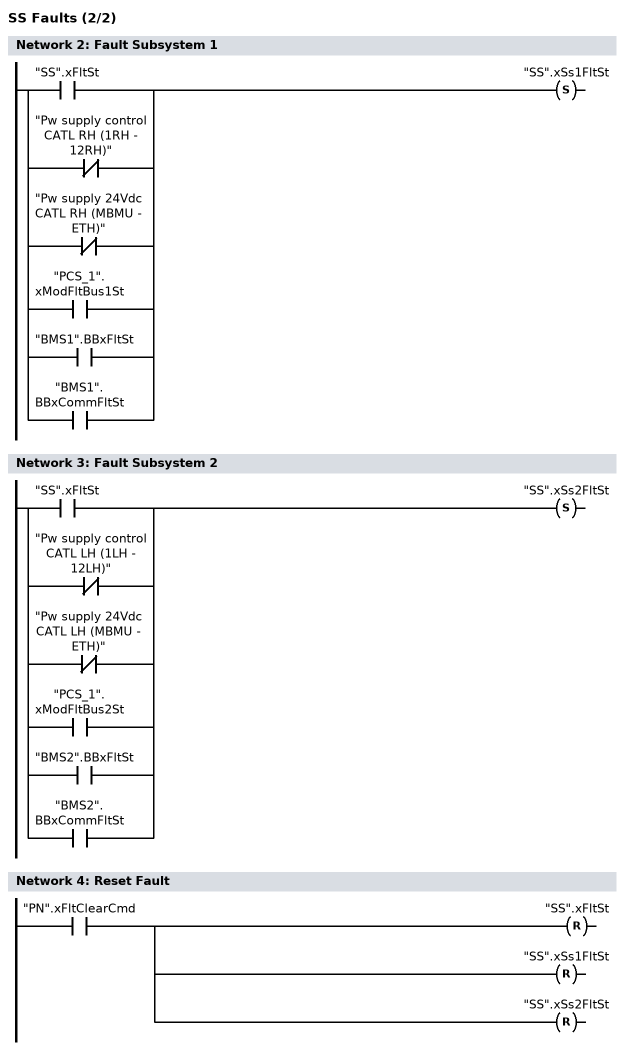
   RUNG wire#powerrail
      Contact( "SS".xFltSt )
      wire#w1
      S_Coil( "SS".xSs1FltSt )
   END_RUNG
   RUNG wire#powerrail
      I_Contact( "Pw supply control CATL RH (1RH - 12RH)" )
   END_RUNG wire#w1
   RUNG wire#powerrail
      I_Contact( "Pw supply 24Vdc CATL RH (MBMU - ETH)" )
   END_RUNG wire#w1
   RUNG wire#powerrail
      Contact( "PCS_1".xModFltBus1St )
   END_RUNG wire#w1
   RUNG wire#powerrail
      Contact( "BMS1".BBxFltSt )
   END_RUNG wire#w1
   RUNG wire#powerrail
      Contact( "BMS1".BBxCommFltSt )
   END_RUNG wire#w1
   // the same network as SCL:
   IF "SS".xFltSt OR NOT "Pw supply control CATL RH (1RH - 12RH)" OR NOT "Pw supply 24Vdc CATL RH (MBMU - ETH)" OR "PCS_1".xModFltBus1St OR "BMS1".BBxFltSt OR "BMS1".BBxCommFltSt THEN
       "SS".xSs1FltSt := TRUE;
   END_IF;
END_REGION

REGION Network 3: Fault Subsystem 2
   RUNG wire#powerrail
      Contact( "SS".xFltSt )
      wire#w1
      S_Coil( "SS".xSs2FltSt )
   END_RUNG
   RUNG wire#powerrail
      I_Contact( "Pw supply control CATL LH (1LH - 12LH)" )
   END_RUNG wire#w1
   RUNG wire#powerrail
      I_Contact( "Pw supply 24Vdc CATL LH (MBMU - ETH)" )
   END_RUNG wire#w1
   RUNG wire#powerrail
      Contact( "PCS_1".xModFltBus2St )
   END_RUNG wire#w1
   RUNG wire#powerrail
      Contact( "BMS2".BBxFltSt )
   END_RUNG wire#w1
   RUNG wire#powerrail
      Contact( "BMS2".BBxCommFltSt )
   END_RUNG wire#w1
   // the same network as SCL:
   IF "SS".xFltSt OR NOT "Pw supply control CATL LH (1LH - 12LH)" OR NOT "Pw supply 24Vdc CATL LH (MBMU - ETH)" OR "PCS_1".xModFltBus2St OR "BMS2".BBxFltSt OR "BMS2".BBxCommFltSt THEN
       "SS".xSs2FltSt := TRUE;
   END_IF;
END_REGION

REGION Network 4: Reset Fault
   RUNG wire#powerrail
      Contact( "PN".xFltClearCmd )
      wire#w1
      R_Coil( "SS".xFltSt )
   END_RUNG
   RUNG wire#w1
      R_Coil( "SS".xSs1FltSt )
   END_RUNG
   RUNG wire#w1
      R_Coil( "SS".xSs2FltSt )
   END_RUNG
   // the same network as SCL:
   IF "PN".xFltClearCmd THEN
       "SS".xFltSt := FALSE;
       "SS".xSs1FltSt := FALSE;
       "SS".xSs2FltSt := FALSE;
   END_IF;
END_REGION
END_FUNCTION

FUNCTION "SS Warnings" : Void   // FC103, LAD
{ S7_Optimized_Access := 'TRUE' }
VERSION : 0.1
// stored: AutoNumber false, IsIECCheckEnabled false, SetENOAutomatically false, UDAEnableTagReadback false
BEGIN

REGION Network 1: Warning Status On/Off
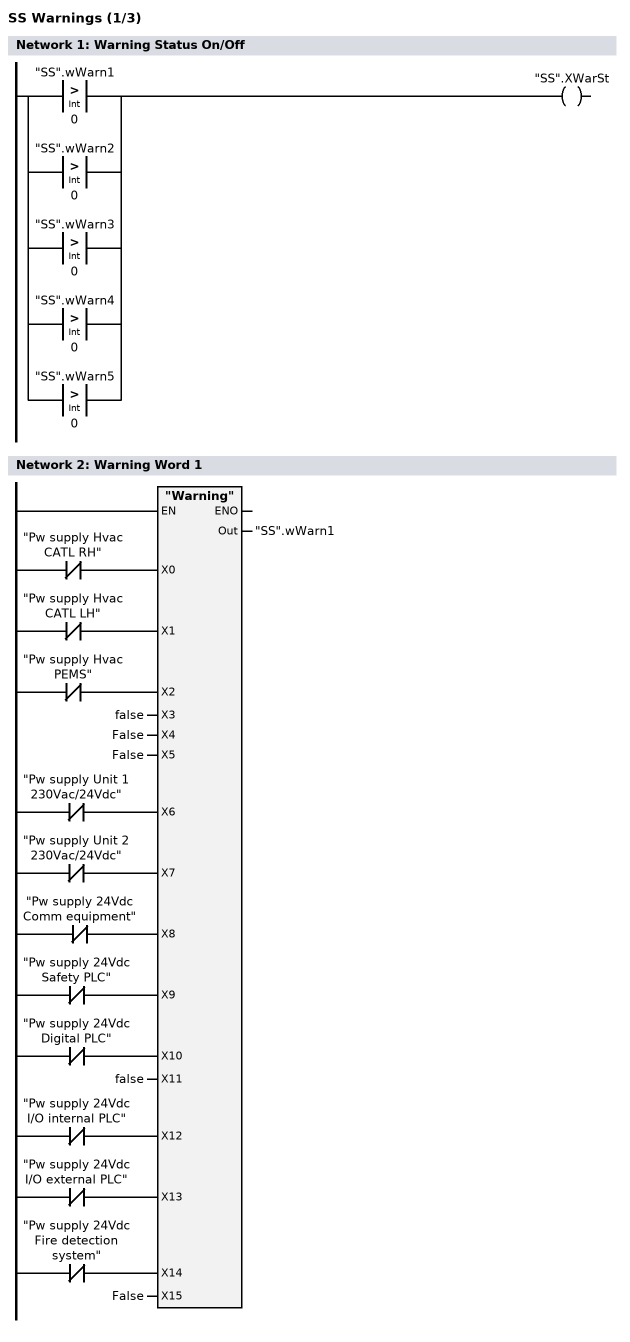
   RUNG wire#powerrail
      { S7_Templates := "SrcType := Int" } GT_Contact(in1 := "SS".wWarn1, in2 := 0)
      wire#w1
      Coil( "SS".XWarSt )
   END_RUNG
   RUNG wire#powerrail
      { S7_Templates := "SrcType := Int" } GT_Contact(in1 := "SS".wWarn2, in2 := 0)
   END_RUNG wire#w1
   RUNG wire#powerrail
      { S7_Templates := "SrcType := Int" } GT_Contact(in1 := "SS".wWarn3, in2 := 0)
   END_RUNG wire#w1
   RUNG wire#powerrail
      { S7_Templates := "SrcType := Int" } GT_Contact(in1 := "SS".wWarn4, in2 := 0)
   END_RUNG wire#w1
   RUNG wire#powerrail
      { S7_Templates := "SrcType := Int" } GT_Contact(in1 := "SS".wWarn5, in2 := 0)
   END_RUNG wire#w1
   // the same network as SCL:
   "SS".XWarSt := ("SS".wWarn1 > 0) OR ("SS".wWarn2 > 0) OR ("SS".wWarn3 > 0) OR ("SS".wWarn4 > 0) OR ("SS".wWarn5 > 0);
END_REGION

REGION Network 2: Warning Word 1
   RUNG wire#powerrail
      "Warning"(X0 := wire#w1, X1 := wire#w2, X2 := wire#w3, X6 := wire#w4, X7 := wire#w5, X8 := wire#w6, X9 := wire#w7, X10 := wire#w8, X12 := wire#w9, X13 := wire#w10, X14 := wire#w11, X3 := false, X4 := False, X5 := False, X11 := false, X15 := False, Out => "SS".wWarn1)
   END_RUNG
   RUNG wire#powerrail
      I_Contact( "Pw supply Hvac CATL RH" )
   END_RUNG wire#w1
   RUNG wire#powerrail
      I_Contact( "Pw supply Hvac CATL LH" )
   END_RUNG wire#w2
   RUNG wire#powerrail
      I_Contact( "Pw supply Hvac PEMS" )
   END_RUNG wire#w3
   RUNG wire#powerrail
      I_Contact( "Pw supply Unit 1 230Vac/24Vdc" )
   END_RUNG wire#w4
   RUNG wire#powerrail
      I_Contact( "Pw supply Unit 2 230Vac/24Vdc" )
   END_RUNG wire#w5
   RUNG wire#powerrail
      I_Contact( "Pw supply 24Vdc Comm equipment" )
   END_RUNG wire#w6
   RUNG wire#powerrail
      I_Contact( "Pw supply 24Vdc Safety PLC" )
   END_RUNG wire#w7
   RUNG wire#powerrail
      I_Contact( "Pw supply 24Vdc Digital PLC" )
   END_RUNG wire#w8
   RUNG wire#powerrail
      I_Contact( "Pw supply 24Vdc I/O internal PLC" )
   END_RUNG wire#w9
   RUNG wire#powerrail
      I_Contact( "Pw supply 24Vdc I/O external PLC" )
   END_RUNG wire#w10
   RUNG wire#powerrail
      I_Contact( "Pw supply 24Vdc Fire detection system" )
   END_RUNG wire#w11
   // the same network as SCL:
   "Warning"(X0 := NOT "Pw supply Hvac CATL RH",
             X1 := NOT "Pw supply Hvac CATL LH",
             X2 := NOT "Pw supply Hvac PEMS",
             X3 := false,
             X4 := False,
             X5 := False,
             X6 := NOT "Pw supply Unit 1 230Vac/24Vdc",
             X7 := NOT "Pw supply Unit 2 230Vac/24Vdc",
             X8 := NOT "Pw supply 24Vdc Comm equipment",
             X9 := NOT "Pw supply 24Vdc Safety PLC",
             X10 := NOT "Pw supply 24Vdc Digital PLC",
             X11 := false,
             X12 := NOT "Pw supply 24Vdc I/O internal PLC",
             X13 := NOT "Pw supply 24Vdc I/O external PLC",
             X14 := NOT "Pw supply 24Vdc Fire detection system",
             X15 := False,
             Out => "SS".wWarn1);
END_REGION

REGION Network 3: Warning Word 2
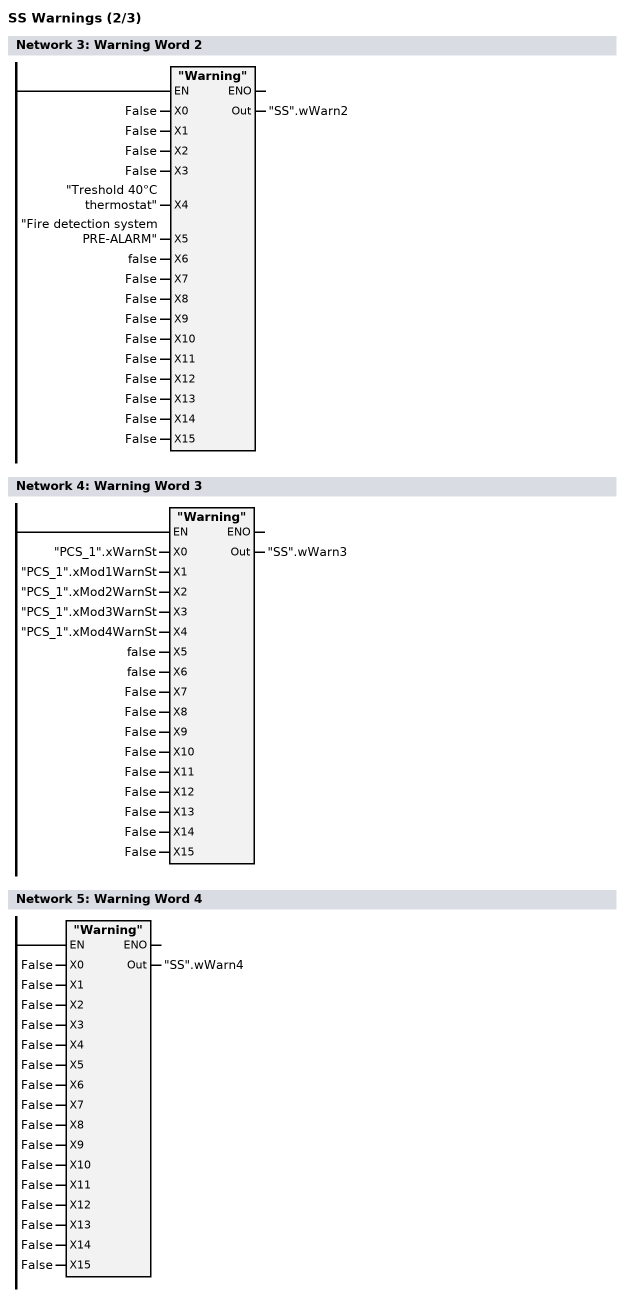
   RUNG wire#powerrail
      "Warning"(X0 := False, X1 := False, X2 := False, X3 := False, X4 := "Treshold 40°C thermostat", X5 := "Fire detection system PRE-ALARM", X6 := false, X7 := False, X8 := False, X9 := False, X10 := False, X11 := False, X12 := False, X13 := False, X14 := False, X15 := False, Out => "SS".wWarn2)
   END_RUNG
   // the same network as SCL:
   "Warning"(X0 := False,
             X1 := False,
             X2 := False,
             X3 := False,
             X4 := "Treshold 40°C thermostat",
             X5 := "Fire detection system PRE-ALARM",
             X6 := false,
             X7 := False,
             X8 := False,
             X9 := False,
             X10 := False,
             X11 := False,
             X12 := False,
             X13 := False,
             X14 := False,
             X15 := False,
             Out => "SS".wWarn2);
END_REGION

REGION Network 4: Warning Word 3
   RUNG wire#powerrail
      "Warning"(X0 := "PCS_1".xWarnSt, X1 := "PCS_1".xMod1WarnSt, X2 := "PCS_1".xMod2WarnSt, X3 := "PCS_1".xMod3WarnSt, X4 := "PCS_1".xMod4WarnSt, X5 := false, X6 := false, X7 := False, X8 := False, X9 := False, X10 := False, X11 := False, X12 := False, X13 := False, X14 := False, X15 := False, Out => "SS".wWarn3)
   END_RUNG
   // the same network as SCL:
   "Warning"(X0 := "PCS_1".xWarnSt,
             X1 := "PCS_1".xMod1WarnSt,
             X2 := "PCS_1".xMod2WarnSt,
             X3 := "PCS_1".xMod3WarnSt,
             X4 := "PCS_1".xMod4WarnSt,
             X5 := false,
             X6 := false,
             X7 := False,
             X8 := False,
             X9 := False,
             X10 := False,
             X11 := False,
             X12 := False,
             X13 := False,
             X14 := False,
             X15 := False,
             Out => "SS".wWarn3);
END_REGION

REGION Network 5: Warning Word 4
   RUNG wire#powerrail
      "Warning"(X0 := False, X1 := False, X2 := False, X3 := False, X4 := False, X5 := False, X6 := False, X7 := False, X8 := False, X9 := False, X10 := False, X11 := False, X12 := False, X13 := False, X14 := False, X15 := False, Out => "SS".wWarn4)
   END_RUNG
   // the same network as SCL:
   "Warning"(X0 := False,
             X1 := False,
             X2 := False,
             X3 := False,
             X4 := False,
             X5 := False,
             X6 := False,
             X7 := False,
             X8 := False,
             X9 := False,
             X10 := False,
             X11 := False,
             X12 := False,
             X13 := False,
             X14 := False,
             X15 := False,
             Out => "SS".wWarn4);
END_REGION

REGION Network 6: Warning Word 5
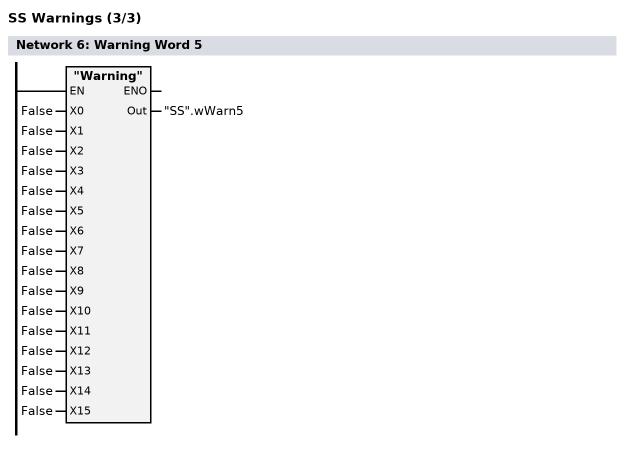
   RUNG wire#powerrail
      "Warning"(X0 := False, X1 := False, X2 := False, X3 := False, X4 := False, X5 := False, X6 := False, X7 := False, X8 := False, X9 := False, X10 := False, X11 := False, X12 := False, X13 := False, X14 := False, X15 := False, Out => "SS".wWarn5)
   END_RUNG
   // the same network as SCL:
   "Warning"(X0 := False,
             X1 := False,
             X2 := False,
             X3 := False,
             X4 := False,
             X5 := False,
             X6 := False,
             X7 := False,
             X8 := False,
             X9 := False,
             X10 := False,
             X11 := False,
             X12 := False,
             X13 := False,
             X14 := False,
             X15 := False,
             Out => "SS".wWarn5);
END_REGION
END_FUNCTION

FUNCTION "Warning" : Void
{ S7_Optimized_Access := 'TRUE' }
VERSION : 0.1
   VAR_INPUT 
      X0 : Bool;
      X1 : Bool;
      X2 : Bool;
      X3 : Bool;
      X4 : Bool;
      X5 : Bool;
      X6 : Bool;
      X7 : Bool;
      X8 : Bool;
      X9 : Bool;
      X10 : Bool;
      X11 : Bool;
      X12 : Bool;
      X13 : Bool;
      X14 : Bool;
      X15 : Bool;
   END_VAR

   VAR_OUTPUT 
      Out : Word;
   END_VAR


BEGIN
	
	#Out.%X0 := #X0;
	#Out.%X1 := #X1;
	#Out.%X2 := #X2;
	#Out.%X3 := #X3;
	#Out.%X4 := #X4;
	#Out.%X5 := #X5;
	#Out.%X6 := #X6;
	#Out.%X7 := #X7;
	#Out.%X8 := #X8;
	#Out.%X9 := #X9;
	#Out.%X10 := #X10;
	#Out.%X11 := #X11;
	#Out.%X12 := #X12;
	#Out.%X13 := #X13;
	#Out.%X14 := #X14;
	#Out.%X15 := #X15;
	
END_FUNCTION

FUNCTION "BMS 1 (F)" : Void   // FC21, LAD
TITLE = ModBus TCP for CATL Battery
{ S7_Optimized_Access := 'TRUE' }
VERSION : 0.1
// stored: AutoNumber false, IsIECCheckEnabled false, SetENOAutomatically false, UDAEnableTagReadback false
   VAR_TEMP
      xSpare : Bool;
      BBwAlm1 : Word;
      BBwWarn1 : Word;
      BR01wAlm1 : Word;
      BR01wAlm2 : Word;
      BR01wAlm3 : Word;
      BR01wWarn1 : Word;
      BR02wAlm1 : Word;
      BR02wAlm2 : Word;
      BR02wAlm3 : Word;
      BR02wWarn1 : Word;
      BR03wAlm1 : Word;
      BR03wAlm2 : Word;
      BR03wAlm3 : Word;
      BR03wWarn1 : Word;
      BR04wAlm1 : Word;
      BR04wAlm2 : Word;
      BR04wAlm3 : Word;
      BR04wWarn1 : Word;
      BR05wAlm1 : Word;
      BR05wAlm2 : Word;
      BR05wAlm3 : Word;
      BR05wWarn1 : Word;
      BR06wAlm1 : Word;
      BR06wAlm2 : Word;
      BR06wAlm3 : Word;
      BR06wWarn1 : Word;
      BR07wAlm1 : Word;
      BR07wAlm2 : Word;
      BR07wAlm3 : Word;
      BR07wWarn1 : Word;
      BR08wAlm1 : Word;
      BR08wAlm2 : Word;
      BR08wAlm3 : Word;
      BR08wWarn1 : Word;
      BR09wAlm1 : Word;
      BR09wAlm2 : Word;
      BR09wAlm3 : Word;
      BR09wWarn1 : Word;
      BR10wAlm1 : Word;
      BR10wAlm2 : Word;
      BR10wAlm3 : Word;
      BR10wWarn1 : Word;
   END_VAR
BEGIN

REGION Network 1: Function Modbus Client
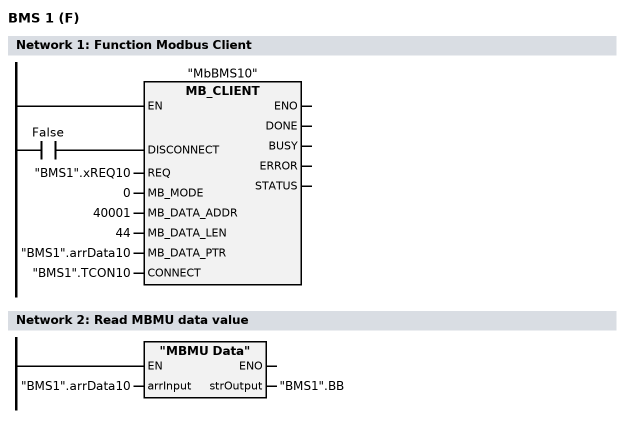
   RUNG wire#powerrail
      "MbBMS10".MB_CLIENT(DISCONNECT := wire#w1, REQ := "BMS1".xREQ10, MB_MODE := 0, MB_DATA_ADDR := 40001, MB_DATA_LEN := 44, MB_DATA_PTR := "BMS1".arrData10, CONNECT := "BMS1".TCON10, DONE =>, BUSY =>, ERROR =>, STATUS =>)
   END_RUNG
   RUNG wire#powerrail
      Contact( False )
   END_RUNG wire#w1
   // the same network as SCL:
   "MbBMS10"(DISCONNECT := False,   // MB_CLIENT
             REQ := "BMS1".xREQ10,
             MB_MODE := 0,
             MB_DATA_ADDR := 40001,
             MB_DATA_LEN := 44,
             MB_DATA_PTR := "BMS1".arrData10,
             CONNECT := "BMS1".TCON10);
END_REGION

REGION Network 2: Read MBMU data value
   RUNG wire#powerrail
      "MBMU Data"(arrInput := "BMS1".arrData10, strOutput => "BMS1".BB)
   END_RUNG
   // the same network as SCL:
   "MBMU Data"(arrInput := "BMS1".arrData10, strOutput => "BMS1".BB);
END_REGION
END_FUNCTION

FUNCTION "MBMU Data" : Void
{ S7_Optimized_Access := 'TRUE' }
VERSION : 0.1
   VAR_INPUT 
      arrInput : Array[1..125] of Word;
   END_VAR

   VAR_OUTPUT 
      strOutput : "BMS_BB";
   END_VAR


BEGIN
	REGION
	    //20210423 First Release
	END_REGION
	
	REGION MBMU Data
	    
	    #strOutput.wWarn1 := #arrInput[1];
	    #strOutput.wWarn2 := #arrInput[2];
	    #strOutput.wWarn3 := #arrInput[3];
	    #strOutput.wWarn4 := #arrInput[4];
	    
	    #strOutput.xInitSt      := #arrInput[17] = 0;
	    #strOutput.xNormOpSt    := #arrInput[17] = 1;
	    #strOutput.xFullChaSt   := #arrInput[17] = 2;
	    #strOutput.xFullDschSt  := #arrInput[17] = 3;
	    #strOutput.xWarnSt      := #arrInput[17] = 4;
	    #strOutput.xFltSt       := #arrInput[17] = 5;
	    
	    #strOutput.rVdcMeas         := INT_TO_REAL(WORD_TO_INT(#arrInput[33])) / 10.0;
	    #strOutput.rIdcMeas         := INT_TO_REAL(WORD_TO_INT(#arrInput[34])) - 20000.0;
	    #strOutput.rSOCmeas         := INT_TO_REAL(WORD_TO_INT(#arrInput[35])) / 10.0;
	    #strOutput.rSOHmeas         := INT_TO_REAL(WORD_TO_INT(#arrInput[36])) / 10.0;
	    #strOutput.rVcellMaxMeas    := INT_TO_REAL(WORD_TO_INT(#arrInput[37])) / 1000.0;
	    #strOutput.rVcellMinMeas    := INT_TO_REAL(WORD_TO_INT(#arrInput[38])) / 1000.0;
	    #strOutput.rVcellAvgMeas    := INT_TO_REAL(WORD_TO_INT(#arrInput[39])) / 1000.0;
	    #strOutput.iTcellMaxMeas    := WORD_TO_INT(#arrInput[40]) - 50;
	    #strOutput.iTcellMinMeas    := WORD_TO_INT(#arrInput[41]) - 50;
	    #strOutput.iTcellAvgMeas    := WORD_TO_INT(#arrInput[42]) - 50;
	    #strOutput.rIchaLim         := INT_TO_REAL(WORD_TO_INT(#arrInput[43])) - 20000.0;
	    #strOutput.rIdschLim        := INT_TO_REAL(WORD_TO_INT(#arrInput[44])) - 20000.0;
	    
	END_REGION
END_FUNCTION

FUNCTION "BMS 1 (M)" : Void   // FC23, LAD
TITLE = ModBus TCP for CATL Battery
{ S7_Optimized_Access := 'TRUE' }
VERSION : 0.1
// stored: AutoNumber false, IsIECCheckEnabled false, SetENOAutomatically false, UDAEnableTagReadback false
   VAR_TEMP
      xSpare : Bool;
      BBwAlm1 : Word;
      BBwWarn1 : Word;
      BR01wAlm1 : Word;
      BR01wAlm2 : Word;
      BR01wAlm3 : Word;
      BR01wWarn1 : Word;
      BR02wAlm1 : Word;
      BR02wAlm2 : Word;
      BR02wAlm3 : Word;
      BR02wWarn1 : Word;
      BR03wAlm1 : Word;
      BR03wAlm2 : Word;
      BR03wAlm3 : Word;
      BR03wWarn1 : Word;
      BR04wAlm1 : Word;
      BR04wAlm2 : Word;
      BR04wAlm3 : Word;
      BR04wWarn1 : Word;
      BR05wAlm1 : Word;
      BR05wAlm2 : Word;
      BR05wAlm3 : Word;
      BR05wWarn1 : Word;
      BR06wAlm1 : Word;
      BR06wAlm2 : Word;
      BR06wAlm3 : Word;
      BR06wWarn1 : Word;
      BR07wAlm1 : Word;
      BR07wAlm2 : Word;
      BR07wAlm3 : Word;
      BR07wWarn1 : Word;
      BR08wAlm1 : Word;
      BR08wAlm2 : Word;
      BR08wAlm3 : Word;
      BR08wWarn1 : Word;
      BR09wAlm1 : Word;
      BR09wAlm2 : Word;
      BR09wAlm3 : Word;
      BR09wWarn1 : Word;
      BR10wAlm1 : Word;
      BR10wAlm2 : Word;
      BR10wAlm3 : Word;
      BR10wWarn1 : Word;
   END_VAR
BEGIN

REGION Network 1: Function Modbus Client
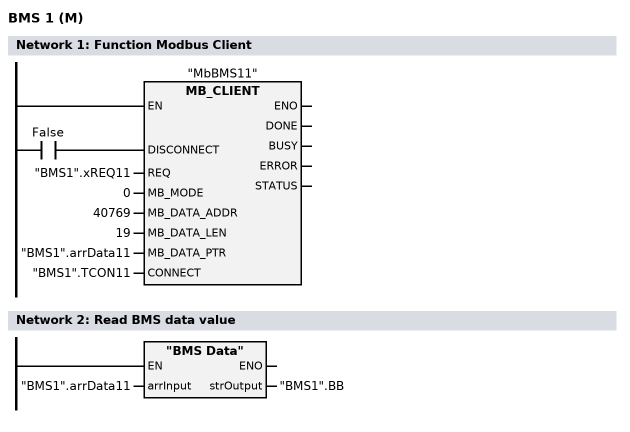
   RUNG wire#powerrail
      "MbBMS11".MB_CLIENT(DISCONNECT := wire#w1, REQ := "BMS1".xREQ11, MB_MODE := 0, MB_DATA_ADDR := 40769, MB_DATA_LEN := 19, MB_DATA_PTR := "BMS1".arrData11, CONNECT := "BMS1".TCON11, DONE =>, BUSY =>, ERROR =>, STATUS =>)
   END_RUNG
   RUNG wire#powerrail
      Contact( False )
   END_RUNG wire#w1
   // the same network as SCL:
   "MbBMS11"(DISCONNECT := False,   // MB_CLIENT
             REQ := "BMS1".xREQ11,
             MB_MODE := 0,
             MB_DATA_ADDR := 40769,
             MB_DATA_LEN := 19,
             MB_DATA_PTR := "BMS1".arrData11,
             CONNECT := "BMS1".TCON11);
END_REGION

REGION Network 2: Read BMS data value
   RUNG wire#powerrail
      "BMS Data"(arrInput := "BMS1".arrData11, strOutput => "BMS1".BB)
   END_RUNG
   // the same network as SCL:
   "BMS Data"(arrInput := "BMS1".arrData11, strOutput => "BMS1".BB);
END_REGION
END_FUNCTION

FUNCTION "BMS Data" : Void
{ S7_Optimized_Access := 'TRUE' }
VERSION : 0.1
   VAR_INPUT 
      arrInput : Array[1..125] of Word;
   END_VAR

   VAR_OUTPUT 
      strOutput : "BMS_BB";
   END_VAR


BEGIN
	REGION
	    // 20210423 First Release
	END_REGION
	
	REGION BMS Data
	    
	    #strOutput.iHeartBeatFb         := WORD_TO_INT(#arrInput[1]);
	    #strOutput.wPwrOnHvSt           := #arrInput[2];
	    #strOutput.wSMstatusSt          := #arrInput[3];
	    #strOutput.iNBRconnectCount     := WORD_TO_INT(#arrInput[5]);
	    #strOutput.rEnergyAvlChaMeas    := INT_TO_REAL(WORD_TO_INT(#arrInput[8])) / 10.0;
	    #strOutput.rEnergyAvlDschMeas   := INT_TO_REAL(WORD_TO_INT(#arrInput[9])) / 10.0;
	    
	END_REGION
END_FUNCTION

FUNCTION "BMS 1 (S)" : Void   // FC25, LAD
TITLE = ModBus TCP for CATL Battery
{ S7_Optimized_Access := 'TRUE' }
VERSION : 0.1
// stored: AutoNumber false, IsIECCheckEnabled false, SetENOAutomatically false, UDAEnableTagReadback false
   VAR_TEMP
      xSpare : Bool;
      BBwAlm1 : Word;
      BBwWarn1 : Word;
      BR01wAlm1 : Word;
      BR01wAlm2 : Word;
      BR01wAlm3 : Word;
      BR01wWarn1 : Word;
      BR02wAlm1 : Word;
      BR02wAlm2 : Word;
      BR02wAlm3 : Word;
      BR02wWarn1 : Word;
      BR03wAlm1 : Word;
      BR03wAlm2 : Word;
      BR03wAlm3 : Word;
      BR03wWarn1 : Word;
      BR04wAlm1 : Word;
      BR04wAlm2 : Word;
      BR04wAlm3 : Word;
      BR04wWarn1 : Word;
      BR05wAlm1 : Word;
      BR05wAlm2 : Word;
      BR05wAlm3 : Word;
      BR05wWarn1 : Word;
      BR06wAlm1 : Word;
      BR06wAlm2 : Word;
      BR06wAlm3 : Word;
      BR06wWarn1 : Word;
      BR07wAlm1 : Word;
      BR07wAlm2 : Word;
      BR07wAlm3 : Word;
      BR07wWarn1 : Word;
      BR08wAlm1 : Word;
      BR08wAlm2 : Word;
      BR08wAlm3 : Word;
      BR08wWarn1 : Word;
      BR09wAlm1 : Word;
      BR09wAlm2 : Word;
      BR09wAlm3 : Word;
      BR09wWarn1 : Word;
      BR10wAlm1 : Word;
      BR10wAlm2 : Word;
      BR10wAlm3 : Word;
      BR10wWarn1 : Word;
      BR11wAlm1 : Word;
      BR11wAlm2 : Word;
      BR11wAlm3 : Word;
      BR11wWarn1 : Word;
      BR12wAlm1 : Word;
      BR12wAlm2 : Word;
      BR12wAlm3 : Word;
      BR12wWarn1 : Word;
   END_VAR
   VAR_TEMP   // added for the SCL form of the ladder/FBD networks
      _w1 : Bool;
   END_VAR
BEGIN

REGION Network 1: Function Modbus Client
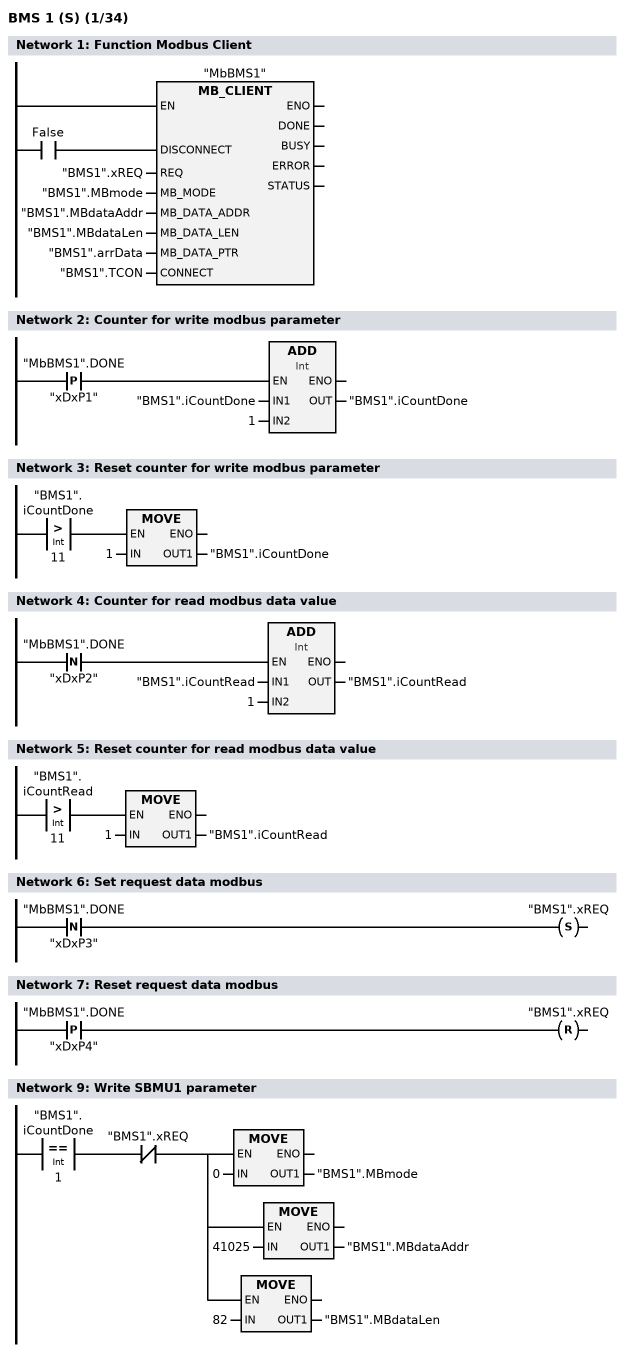
   RUNG wire#powerrail
      "MbBMS1".MB_CLIENT(DISCONNECT := wire#w1, REQ := "BMS1".xREQ, MB_MODE := "BMS1".MBmode, MB_DATA_ADDR := "BMS1".MBdataAddr, MB_DATA_LEN := "BMS1".MBdataLen, MB_DATA_PTR := "BMS1".arrData, CONNECT := "BMS1".TCON, DONE =>, BUSY =>, ERROR =>, STATUS =>)
   END_RUNG
   RUNG wire#powerrail
      Contact( False )
   END_RUNG wire#w1
   // the same network as SCL:
   "MbBMS1"(DISCONNECT := False,   // MB_CLIENT
            REQ := "BMS1".xREQ,
            MB_MODE := "BMS1".MBmode,
            MB_DATA_ADDR := "BMS1".MBdataAddr,
            MB_DATA_LEN := "BMS1".MBdataLen,
            MB_DATA_PTR := "BMS1".arrData,
            CONNECT := "BMS1".TCON);
END_REGION

REGION Network 2: Counter for write modbus parameter
   RUNG wire#powerrail
      P_Contact(operand := "MbBMS1".DONE, bit := "xDxP1")
      { S7_Templates := "SrcType := Int" } Add(in1 := "BMS1".iCountDone, in2 := 1, out => "BMS1".iCountDone)
   END_RUNG
   // the same network as SCL:
   #_w1 := "MbBMS1".DONE AND NOT "xDxP1";   // rising edge of "MbBMS1".DONE
   "xDxP1" := "MbBMS1".DONE;
   IF #_w1 THEN "BMS1".iCountDone := "BMS1".iCountDone + 1; END_IF;
END_REGION

REGION Network 3: Reset counter for write modbus parameter
   RUNG wire#powerrail
      { S7_Templates := "SrcType := Int" } GT_Contact(in1 := "BMS1".iCountDone, in2 := 11)
      Move(in := 1, out1 => "BMS1".iCountDone)
   END_RUNG
   // the same network as SCL:
   IF "BMS1".iCountDone > 11 THEN "BMS1".iCountDone := 1; END_IF;
END_REGION

REGION Network 4: Counter for read modbus data value
   RUNG wire#powerrail
      N_Contact(operand := "MbBMS1".DONE, bit := "xDxP2")
      { S7_Templates := "SrcType := Int" } Add(in1 := "BMS1".iCountRead, in2 := 1, out => "BMS1".iCountRead)
   END_RUNG
   // the same network as SCL:
   #_w1 := NOT "MbBMS1".DONE AND "xDxP2";   // falling edge of "MbBMS1".DONE
   "xDxP2" := "MbBMS1".DONE;
   IF #_w1 THEN "BMS1".iCountRead := "BMS1".iCountRead + 1; END_IF;
END_REGION

REGION Network 5: Reset counter for read modbus data value
   RUNG wire#powerrail
      { S7_Templates := "SrcType := Int" } GT_Contact(in1 := "BMS1".iCountRead, in2 := 11)
      Move(in := 1, out1 => "BMS1".iCountRead)
   END_RUNG
   // the same network as SCL:
   IF "BMS1".iCountRead > 11 THEN "BMS1".iCountRead := 1; END_IF;
END_REGION

REGION Network 6: Set request data modbus
   RUNG wire#powerrail
      N_Contact(operand := "MbBMS1".DONE, bit := "xDxP3")
      S_Coil( "BMS1".xREQ )
   END_RUNG
   // the same network as SCL:
   #_w1 := NOT "MbBMS1".DONE AND "xDxP3";   // falling edge of "MbBMS1".DONE
   "xDxP3" := "MbBMS1".DONE;
   IF #_w1 THEN "BMS1".xREQ := TRUE; END_IF;
END_REGION

REGION Network 7: Reset request data modbus
   RUNG wire#powerrail
      P_Contact(operand := "MbBMS1".DONE, bit := "xDxP4")
      R_Coil( "BMS1".xREQ )
   END_RUNG
   // the same network as SCL:
   #_w1 := "MbBMS1".DONE AND NOT "xDxP4";   // rising edge of "MbBMS1".DONE
   "xDxP4" := "MbBMS1".DONE;
   IF #_w1 THEN "BMS1".xREQ := FALSE; END_IF;
END_REGION

REGION Network 9: Write SBMU1 parameter
   RUNG wire#powerrail
      { S7_Templates := "SrcType := Int" } EQ_Contact(in1 := "BMS1".iCountDone, in2 := 1)
      I_Contact( "BMS1".xREQ )
      wire#w1
      Move(in := 0, out1 => "BMS1".MBmode)
   END_RUNG
   RUNG wire#w1
      Move(in := 41025, out1 => "BMS1".MBdataAddr)
   END_RUNG
   RUNG wire#w1
      Move(in := 82, out1 => "BMS1".MBdataLen)
   END_RUNG
   // the same network as SCL:
   IF ("BMS1".iCountDone = 1) AND NOT "BMS1".xREQ THEN
       "BMS1".MBmode := 0;
       "BMS1".MBdataAddr := 41025;
       "BMS1".MBdataLen := 82;
   END_IF;
END_REGION

REGION Network 10: Read SBMU1 data value
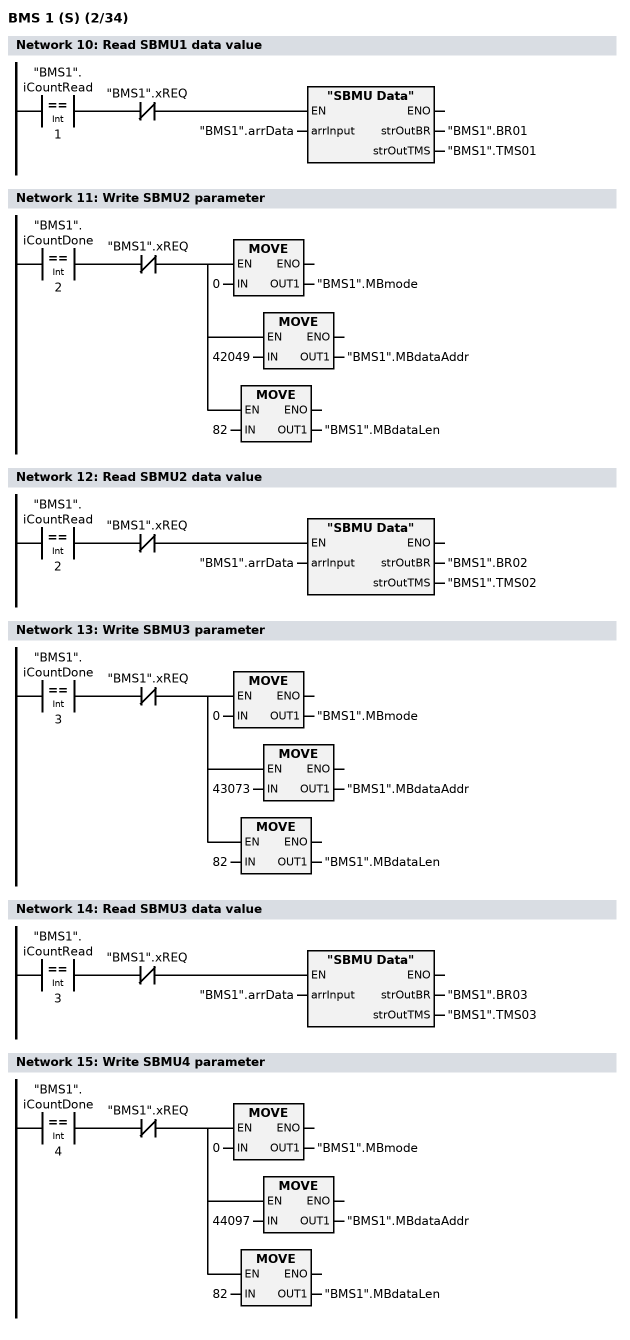
   RUNG wire#powerrail
      { S7_Templates := "SrcType := Int" } EQ_Contact(in1 := "BMS1".iCountRead, in2 := 1)
      I_Contact( "BMS1".xREQ )
      "SBMU Data"(arrInput := "BMS1".arrData, strOutBR => "BMS1".BR01, strOutTMS => "BMS1".TMS01)
   END_RUNG
   // the same network as SCL:
   IF ("BMS1".iCountRead = 1) AND NOT "BMS1".xREQ THEN
       "SBMU Data"(arrInput := "BMS1".arrData, strOutBR => "BMS1".BR01, strOutTMS => "BMS1".TMS01);
   END_IF;
END_REGION

REGION Network 11: Write SBMU2 parameter
   RUNG wire#powerrail
      { S7_Templates := "SrcType := Int" } EQ_Contact(in1 := "BMS1".iCountDone, in2 := 2)
      I_Contact( "BMS1".xREQ )
      wire#w1
      Move(in := 0, out1 => "BMS1".MBmode)
   END_RUNG
   RUNG wire#w1
      Move(in := 42049, out1 => "BMS1".MBdataAddr)
   END_RUNG
   RUNG wire#w1
      Move(in := 82, out1 => "BMS1".MBdataLen)
   END_RUNG
   // the same network as SCL:
   IF ("BMS1".iCountDone = 2) AND NOT "BMS1".xREQ THEN
       "BMS1".MBmode := 0;
       "BMS1".MBdataAddr := 42049;
       "BMS1".MBdataLen := 82;
   END_IF;
END_REGION

REGION Network 12: Read SBMU2 data value
   RUNG wire#powerrail
      { S7_Templates := "SrcType := Int" } EQ_Contact(in1 := "BMS1".iCountRead, in2 := 2)
      I_Contact( "BMS1".xREQ )
      "SBMU Data"(arrInput := "BMS1".arrData, strOutBR => "BMS1".BR02, strOutTMS => "BMS1".TMS02)
   END_RUNG
   // the same network as SCL:
   IF ("BMS1".iCountRead = 2) AND NOT "BMS1".xREQ THEN
       "SBMU Data"(arrInput := "BMS1".arrData, strOutBR => "BMS1".BR02, strOutTMS => "BMS1".TMS02);
   END_IF;
END_REGION

